            Host_Computer.StagingA_L2_ErrorCode := 0;
            Host_Computer.StagingA_L2_Retryable := FALSE;
            Host_Computer.StagingA_L2_CompletedSeq := Host_Computer.StagingA_L2_AcceptedSeq;
            Host_Computer.StagingA_L2_Step := 99;
            Host_Computer.StagingA_L2_State := 20;

        ELSE
            Host_Computer.StagingA_L2_ErrorCode := 103;
            Host_Computer.StagingA_L2_Retryable := FALSE;
            Host_Computer.StagingA_L2_CompletedSeq := Host_Computer.StagingA_L2_AcceptedSeq;
            Host_Computer.StagingA_L2_State := 40;
    END_CASE
END_IF

// 上位机看到终态后会清 Start=FALSE，并等待 State 回 IDLE。
// 保留 CompletedSeq，不清它，否则上位机会丢失已完成序号。
IF NOT Host_Computer.StagingA_L2_Start THEN
    IF (Host_Computer.StagingA_L2_State = 20)
    OR (Host_Computer.StagingA_L2_State = 30)
    OR (Host_Computer.StagingA_L2_State = 40)
    OR (Host_Computer.StagingA_L2_State = 50) THEN
        Host_Computer.StagingA_L2_State := 0;
        Host_Computer.StagingA_L2_ActiveCode := 0;
        Host_Computer.StagingA_L2_Step := 0;
        Host_Computer.StagingA_L2_ErrorCode := 0;
        Host_Computer.StagingA_L2_SafeState := 0;
        Host_Computer.StagingA_L2_Retryable := FALSE;
    END_IF
END_IF

END_PROGRAM

// Device/Application/50_action/Rail_L2
PROGRAM Rail_L2
VAR
	L2_StartTrig : R_TRIG;
	fTgt: LREAL;
END_VAR

(* 地轨 11Y L2 统一动作派发器 (第7通道).
   按位置码移地轨: Rail_L2_ActionCode=10 -> 移到 Rail_Pos_Target[Rail_Target_Position] (1..6, PC 真源).
   地轨坐标真源已收编为 PC 写的 Rail_Pos_Target[]; HMI position[] 降为手动示教工作副本, 自动不再读它.
   Start 上升沿接受 -> RUNNING 下发移动 -> bAbMoveDone=DONE. *)
L2_StartTrig(CLK := Rail_L2_Start);

(* Global deployment/startup gate: reject before any physical action is dispatched. *)
IF L2_StartTrig.Q AND (Rail_L2_State=0)
	AND ((NOT PLC_Ready) OR (PLC_Deploy_State<>0)) THEN
	Rail_L2_AcceptedSeq := Rail_L2_RequestSeq;
	Rail_L2_ActiveCode := Rail_L2_ActionCode;
	Rail_L2_ErrorCode := 190;
	Rail_L2_Retryable := TRUE;
	Rail_L2_CompletedSeq := Rail_L2_RequestSeq;
	Rail_L2_State := 30;
	RETURN;
END_IF

CASE Rail_L2_State OF
	0:  (* IDLE *)
		Rail_L2_Step := 0;
		IF L2_StartTrig.Q THEN
			Rail_L2_AcceptedSeq := Rail_L2_RequestSeq;
			Rail_L2_ActiveCode  := Rail_L2_ActionCode;
			Rail_L2_ErrorCode   := 0;
			Rail_L2_Retryable   := FALSE;
// 			IF Rail_L2_ActionCode = 10
// 			   AND Rail_Target_Position >= 1 AND Rail_Target_Position <= 6 THEN
// 				Rail_L2_SafeState := 0;
// // 				地轨轴11YDATE.fAbsTarget := HMI_地轨轴11Y.position[Rail_Target_Position];
// 				地轨轴11YDATE.fAbsTarget := Rail_Pos_Target[Rail_Target_Position];
// 				地轨轴11YDATE.xMoveAbs   := TRUE;
// 				Rail_L2_State := 10;   (* RUNNING *)
// 			ELSE
// 				Rail_L2_ErrorCode    := 101;  (* 未知动作码 / 非法位置码 *)
// 				Rail_L2_Retryable    := TRUE;
// 				Rail_L2_CompletedSeq := Rail_L2_AcceptedSeq;
// 				Rail_L2_State        := 30;   (* REJECTED *)
// 			END_IF
			IF Rail_L2_ActionCode = 10 AND Rail_Target_Position >= 1 AND Rail_Target_Position <= 6 THEN
				fTgt := Rail_Pos_Target[Rail_Target_Position];     (* PC 真源坐标 *)
				IF fTgt <= 0.0 OR fTgt > 3000.0 THEN
					(* 兜底: PC 未 push / 重启后 Rail_Pos_Target 归 0 / 越限 → 拒绝, 绝不移到 0 端 *)
					Rail_L2_ErrorCode    := 102;   (* 目标未初始化或越限 *)
					Rail_L2_Retryable    := TRUE;
					Rail_L2_CompletedSeq := Rail_L2_AcceptedSeq;
					Rail_L2_State        := 30;    (* REJECTED *)
				ELSE
					Rail_L2_SafeState        := 0;
					地轨轴11YDATE.fAbsTarget := fTgt;
					地轨轴11YDATE.xMoveAbs   := TRUE;
					Rail_L2_State            := 10; (* RUNNING *)
				END_IF
			ELSE
				Rail_L2_ErrorCode    := 101;   (* 未知动作码 / 非法位置码 *)
				Rail_L2_Retryable    := TRUE;
				Rail_L2_CompletedSeq := Rail_L2_AcceptedSeq;
				Rail_L2_State        := 30;    (* REJECTED *)
END_IF
		END_IF

	10: (* RUNNING *)
		IF Rail_L2_Reset THEN                 (* RUNNING 中 RESET: 中止回 IDLE *)
			地轨轴11YDATE.xMoveAbs := FALSE;
			Rail_L2_State := 0;
		ELSIF 地轨轴11YDATE.bAbMoveDone THEN
			地轨轴11YDATE.xMoveAbs   := FALSE;
			Rail_L2_CompletedSeq := Rail_L2_AcceptedSeq;
			Rail_L2_State        := 20;   (* DONE *)
		END_IF
		(* 如地轨伺服有报警位, 在此 ELSIF <报警> THEN 置 Rail_L2_ErrorCode + State:=40 *)

	20, 30, 40, 50:  (* 终态: 等 Start 落沿或 Reset 回 IDLE *)
		IF (NOT Rail_L2_Start) OR Rail_L2_Reset THEN
			Rail_L2_State := 0;
		END_IF
END_CASE

END_PROGRAM

// Device/Application/50_action/FeedLift_L2
PROGRAM FeedLift_L2
VAR
	初始化step: INT;
	上料step: INT;
	下料step: INT;
	bActionDone: BOOL;
	bActionError: BOOL;
	L2_StartTrig: R_TRIG;
	feedlift_TO: TON;
	FeedLift_1Z_RaiseRetryCount : INT;
	FeedLift_1Z_RaiseStartPos   : LREAL;
	FeedLift_1Z_ClearRetryCount : INT;
	FeedLift_1Z_ClearStartPos   : LREAL;
	FeedLift_2Z_ReadyRetryCount : INT;
	FeedLift_2Z_ReadyStartPos   : LREAL;
	FeedLift_2Z_BuryRetryCount  : INT;
	FeedLift_2Z_BuryStartPos    : LREAL;
END_VAR

(* FeedLift 工位 L2 统一动作派发器
   按 FeedLift_L2_ActionCode 派发到纯设备原子动作 (不含机器人/相机/CNC 握手).
   Start 上升沿接受请求 -> RUNNING 每周期调用对应原子 -> bActionDone=DONE / bActionError=ERROR. *)
L2_StartTrig(CLK := FeedLift_L2_Start);

(* Global deployment/startup gate: reject before any physical action is dispatched. *)
IF L2_StartTrig.Q AND (FeedLift_L2_State=0)
	AND ((NOT PLC_Ready) OR (PLC_Deploy_State<>0)) THEN
	FeedLift_L2_AcceptedSeq := FeedLift_L2_RequestSeq;
	FeedLift_L2_ActiveCode := FeedLift_L2_ActionCode;
	FeedLift_L2_ErrorCode := 190;
	FeedLift_L2_Retryable := TRUE;
	FeedLift_L2_CompletedSeq := FeedLift_L2_RequestSeq;
	FeedLift_L2_State := 30;
	RETURN;
END_IF

CASE FeedLift_L2_State OF
	0:  (* IDLE *)
		FeedLift_L2_Step := 0;
		IF L2_StartTrig.Q THEN
			FeedLift_L2_AcceptedSeq := FeedLift_L2_RequestSeq;
			FeedLift_L2_ActiveCode  := FeedLift_L2_ActionCode;
			FeedLift_L2_ErrorCode   := 0;
			FeedLift_L2_Retryable   := FALSE;
			bActionDone  := FALSE;
			bActionError := FALSE;
			初始化step := 0;
			上料step := 0;
			下料step := 0;
			CASE FeedLift_L2_ActionCode OF
				10, 11, 12, 13, 21, 22, 91:
					FeedLift_L2_SafeState := 0;
					FeedLift_L2_State     := 10;   (* RUNNING *)
			ELSE
				FeedLift_L2_ErrorCode    := 101;  (* 未知动作码 *)
				FeedLift_L2_Retryable    := TRUE;
				FeedLift_L2_CompletedSeq := FeedLift_L2_AcceptedSeq;
				FeedLift_L2_State        := 30;   (* REJECTED *)
			END_CASE
		END_IF

	10: (* RUNNING *)
		IF FeedLift_L2_Reset THEN FeedLift_L2_State := 0; RETURN; END_IF   (* RUNNING 中 RESET: 中止挂死动作 *)
		CASE FeedLift_L2_ActiveCode OF
			10: A10_init_初始化();
			11: A11_feed_raise();
			12: A12_feed_lower();
			13: A13_feed_clear();
			21: A21_unload_ready();
			22: A22_unload_bury();
			91: A91_endcheck();
		END_CASE
		IF bActionDone THEN
			bActionDone              := FALSE;
			FeedLift_L2_CompletedSeq := FeedLift_L2_AcceptedSeq;
			FeedLift_L2_State        := 20;   (* DONE *)
		ELSIF bActionError THEN              (* 设备预条件未满足 -> 报错交上位机 *)
			bActionError             := FALSE;
			FeedLift_L2_Retryable    := TRUE;
			FeedLift_L2_CompletedSeq := FeedLift_L2_AcceptedSeq;
			FeedLift_L2_State        := 40;   (* ERROR; ErrorCode 由原子置 *)
		END_IF

	20, 30, 40, 50:  (* 终态: 等 Start 落沿或 Reset 回 IDLE *)
		IF (NOT FeedLift_L2_Start) OR FeedLift_L2_Reset THEN
			FeedLift_L2_State := 0;
		END_IF
END_CASE

ACTION A11_feed_raise:
(* FeedLift feed_raise: bounded 1Z jog; final PE1 stable TRUE *)
// CASE 上料step OF
// 	0:
// 		Z1JOG_pos:=FALSE;
// 		feedlift_TO(IN:=FALSE, PT:=T#200MS);
// 		IF FeedLift_1Z_SearchLowTarget >= FeedLift_1Z_SearchHighTarget THEN
// 			FeedLift_L2_ErrorCode:=303;
// 			上料step:=0;
// 			bActionError:=TRUE;
// 		ELSIF 玻璃上料轴1ZDATE.bHomed AND 玻璃升降接近开关1 AND 上料进料传感器 AND NOT Alarm.0 THEN
// 			上料step:=10;
// 		ELSE
// 			feedlift_TO(IN:=TRUE, PT:=T#10S);
// 			IF feedlift_TO.Q THEN
// 				FeedLift_L2_ErrorCode:=301;
// 				上料step:=0;
// 				bActionError:=TRUE;
// 			END_IF
// 		END_IF
// 	10:
// 		feedlift_TO(IN:=FALSE, PT:=T#200MS);
// 		IF 玻璃升降光电开关1 THEN
// 			Z1JOG_pos:=FALSE;
// 			上料step:=20;
// 		ELSIF 玻璃上料轴1ZDATE.fActPos < FeedLift_1Z_SearchHighTarget THEN
// 			Z1JOG_pos:=TRUE;
// 		ELSE
// 			Z1JOG_pos:=FALSE;
// 			FeedLift_L2_ErrorCode:=304;
// 			上料step:=0;
// 			bActionError:=TRUE;
// 		END_IF
// 	20:
// 		Z1JOG_pos:=FALSE;
// 		feedlift_TO(IN:=玻璃升降光电开关1, PT:=T#200MS);
// 		IF feedlift_TO.Q THEN
// 			上料step:=0;
// 			bActionDone:=TRUE;
// 		ELSIF NOT 玻璃升降光电开关1 THEN
// 			IF 玻璃上料轴1ZDATE.fActPos < FeedLift_1Z_SearchHighTarget THEN
// 				上料step:=10;
// 			ELSE
// 				FeedLift_L2_ErrorCode:=304;
// 				上料step:=0;
// 				bActionError:=TRUE;
// 			END_IF
// 		END_IF
// END_CASE

(* FeedLift feed_raise:
   目标是找到并停在 1Z 上料取料位: 玻璃升降光电开关1 = TRUE。
   - 启动时已 TRUE: 原地停住, 稳定确认 DONE。
   - 启动时 FALSE: 只向上搜索 TRUE。
   - 看到 TRUE 后先停住, 再计时确认。
   - 确认中抖成 FALSE: 只向上小幅重捕获。
   - 失败用 304, 通过 FeedLift_L2_Step 区分阶段。 *)
CASE 上料step OF
	0:
		FeedLift_L2_Step := 11;  (* 初始化 / 前置检查 *)
		Z1JOG_pos := FALSE;
		feedlift_TO(IN := FALSE, PT := T#300MS);
		FeedLift_1Z_RaiseRetryCount := 0;
		FeedLift_1Z_RaiseStartPos := 玻璃上料轴1ZDATE.fActPos;

		IF FeedLift_1Z_SearchLowTarget >= FeedLift_1Z_SearchHighTarget THEN
			FeedLift_L2_ErrorCode := 303;
			上料step := 0;
			bActionError := TRUE;
		ELSE
			上料step := 5;
		END_IF

	5:
		FeedLift_L2_Step := 11;  (* 等待前置条件满足 *)
		Z1JOG_pos := FALSE;

		IF 玻璃上料轴1ZDATE.bHomed AND 玻璃升降接近开关1 AND 上料进料传感器 AND NOT Alarm.0 THEN
			feedlift_TO(IN := FALSE, PT := T#300MS);
			IF 玻璃升降光电开关1 THEN
				上料step := 20;
			ELSE
				上料step := 10;
			END_IF
		ELSE
			feedlift_TO(IN := TRUE, PT := T#10S);
			IF feedlift_TO.Q THEN
				FeedLift_L2_ErrorCode := 301;
				上料step := 0;
				bActionError := TRUE;
			END_IF
		END_IF

	10:
		FeedLift_L2_Step := 11;  (* 向上搜索 TRUE *)
		feedlift_TO(IN := FALSE, PT := T#300MS);

		IF 玻璃升降光电开关1 THEN
			Z1JOG_pos := FALSE;
			上料step := 20;
		ELSIF 玻璃上料轴1ZDATE.fActPos < FeedLift_1Z_SearchHighTarget THEN
			Z1JOG_pos := TRUE;
		ELSE
			Z1JOG_pos := FALSE;
			FeedLift_L2_Step := 14;  (* 失败收敛 *)
			FeedLift_L2_ErrorCode := 304;
			上料step := 0;
			bActionError := TRUE;
		END_IF

	20:
		FeedLift_L2_Step := 12;  (* 停住后确认 TRUE 稳定 *)
		Z1JOG_pos := FALSE;
		feedlift_TO(IN := 玻璃升降光电开关1, PT := T#300MS);

		IF feedlift_TO.Q THEN
			上料step := 0;
			bActionDone := TRUE;
		ELSIF NOT 玻璃升降光电开关1 THEN
			feedlift_TO(IN := FALSE, PT := T#300MS);
			IF FeedLift_1Z_RaiseRetryCount < 2 THEN
				FeedLift_1Z_RaiseRetryCount := FeedLift_1Z_RaiseRetryCount + 1;
				FeedLift_1Z_RaiseStartPos := 玻璃上料轴1ZDATE.fActPos;
				上料step := 30;
			ELSE
				FeedLift_L2_Step := 14;  (* 失败收敛 *)
				FeedLift_L2_ErrorCode := 304;
				上料step := 0;
				bActionError := TRUE;
			END_IF
		END_IF

	30:
		FeedLift_L2_Step := 13;  (* 小幅向上重捕获 TRUE *)
		feedlift_TO(IN := FALSE, PT := T#300MS);

		IF 玻璃升降光电开关1 THEN
			Z1JOG_pos := FALSE;
			上料step := 20;
		ELSIF 玻璃上料轴1ZDATE.fActPos >= FeedLift_1Z_SearchHighTarget THEN
			Z1JOG_pos := FALSE;
			FeedLift_L2_Step := 14;  (* 失败收敛 *)
			FeedLift_L2_ErrorCode := 304;
			上料step := 0;
			bActionError := TRUE;
		ELSIF (玻璃上料轴1ZDATE.fActPos - FeedLift_1Z_RaiseStartPos) >= 2.0 THEN
			Z1JOG_pos := FALSE;
			FeedLift_L2_Step := 14;  (* 失败收敛 *)
			FeedLift_L2_ErrorCode := 304;
			上料step := 0;
			bActionError := TRUE;
		ELSE
			Z1JOG_pos := TRUE;
		END_IF
END_CASE
END_ACTION

ACTION A10_init_初始化:
(* FeedLift init:
   清 L2 域内的残留命令位, 再校验 1Z/2Z 已回零。
   - jog 位: 任一搜索动作被 L2_Reset 中止时会停在 TRUE, 不清则下次上电即自行走轴。
   - xMoveRel: A12_feed_lower 在 step0 置位、step10 才清, 中途 Reset 同样留 TRUE。
   - 步序变量由派发器 IDLE 受理时统一清零, 此处不重复。
   本动作不产生任何轴运动: 双轴回零只能在 HMI 按【一键回原点】, 上位机无此通道,
   故未回零时只报 308 交上位机, 不自行 Home。
   失败用 308, 通过 FeedLift_L2_Step 区分阶段。 *)
CASE 初始化step OF
	0:
		FeedLift_L2_Step := 51;  (* 清残留命令位 *)
		Z1JOG_pos := FALSE;
		Z1JOG_neg := FALSE;
		Z2JOG_POS := FALSE;
		Z2JOG_NEG := FALSE;
		玻璃上料轴1ZDATE.xMoveRel := FALSE;
		玻璃上料轴2ZDATE.xMoveRel := FALSE;
		feedlift_TO(IN := FALSE, PT := T#300MS);
		初始化step := 10;

	10:
		FeedLift_L2_Step := 52;  (* 校验双轴已回零 *)
		IF 玻璃上料轴1ZDATE.bHomed AND 玻璃上料轴2ZDATE.bHomed THEN
			初始化step := 0;
			bActionDone := TRUE;
		ELSE
			feedlift_TO(IN := TRUE, PT := T#5S);
			IF feedlift_TO.Q THEN
				FeedLift_L2_Step := 54;  (* 失败收敛 *)
				FeedLift_L2_ErrorCode := 308;
				初始化step := 0;
				bActionError := TRUE;
			END_IF
		END_IF
END_CASE
END_ACTION

ACTION A22_unload_bury:
(* FeedLift unload_bury: bounded 2Z jog to make PE2 stable FALSE; reverse once if low misses *)
// CASE 下料step OF
// 	0:
// 		Z2JOG_POS:=FALSE;
// 		Z2JOG_NEG:=FALSE;
// 		feedlift_TO(IN:=FALSE, PT:=T#200MS);
// 		IF FeedLift_2Z_SearchLowTarget >= FeedLift_2Z_SearchHighTarget THEN
// 			FeedLift_L2_ErrorCode:=303;
// 			下料step:=0;
// 			bActionError:=TRUE;
// 		ELSIF 玻璃升降光电开关2 AND 玻璃升降接近开关2 THEN
// 			下料step:=10;
// 		ELSE
// 			feedlift_TO(IN:=TRUE, PT:=T#10S);
// 			IF feedlift_TO.Q THEN
// 				FeedLift_L2_ErrorCode:=302;
// 				下料step:=0;
// 				bActionError:=TRUE;
// 			END_IF
// 		END_IF
// 	10:
// 		Z2JOG_POS:=FALSE;
// 		IF NOT 玻璃升降光电开关2 THEN
// 			Z2JOG_NEG:=FALSE;
// 			下料step:=30;
// 		ELSIF 玻璃上料轴2ZDATE.fActPos > FeedLift_2Z_SearchLowTarget THEN
// 			Z2JOG_NEG:=TRUE;
// 		ELSE
// 			Z2JOG_NEG:=FALSE;
// 			下料step:=20;
// 		END_IF
// 	20:
// 		Z2JOG_NEG:=FALSE;
// 		IF NOT 玻璃升降光电开关2 THEN
// 			Z2JOG_POS:=FALSE;
// 			下料step:=30;
// 		ELSIF 玻璃上料轴2ZDATE.fActPos < FeedLift_2Z_SearchHighTarget THEN
// 			Z2JOG_POS:=TRUE;
// 		ELSE
// 			Z2JOG_POS:=FALSE;
// 			FeedLift_L2_ErrorCode:=305;
// 			下料step:=0;
// 			bActionError:=TRUE;
// 		END_IF
// 	30:
// 		Z2JOG_POS:=FALSE;
// 		Z2JOG_NEG:=FALSE;
// 		feedlift_TO(IN:=NOT 玻璃升降光电开关2, PT:=T#200MS);
// 		IF feedlift_TO.Q THEN
// 			下料step:=0;
// 			bActionDone:=TRUE;
// 		ELSIF 玻璃升降光电开关2 THEN
// 			IF 玻璃上料轴2ZDATE.fActPos > FeedLift_2Z_SearchLowTarget THEN
// 				下料step:=10;
// 			ELSIF 玻璃上料轴2ZDATE.fActPos < FeedLift_2Z_SearchHighTarget THEN
// 				下料step:=20;
// 			ELSE
// 				FeedLift_L2_ErrorCode:=305;
// 				下料step:=0;
// 				bActionError:=TRUE;
// 			END_IF
// 		END_IF
// END_CASE

(* FeedLift unload_bury:
   目标是机器人放废板后, 2Z 向下埋料直到 玻璃升降光电开关2 = FALSE。
   - 启动时已 FALSE: 原地停住, 稳定确认 DONE。
   - 启动时 TRUE: 只向下搜索 FALSE。
   - 看到 FALSE 后先停住, 再计时确认。
   - 确认中抖成 TRUE: 只向下小幅重捕获, 不反向上扫。
   - 失败用 305, 通过 FeedLift_L2_Step 区分阶段。 *)
CASE 下料step OF
	0:
		FeedLift_L2_Step := 31;  (* 初始化 / 前置检查 *)
		Z2JOG_POS := FALSE;
		Z2JOG_NEG := FALSE;
		feedlift_TO(IN := FALSE, PT := T#300MS);
		FeedLift_2Z_BuryRetryCount := 0;
		FeedLift_2Z_BuryStartPos := 玻璃上料轴2ZDATE.fActPos;

		IF FeedLift_2Z_SearchLowTarget >= FeedLift_2Z_SearchHighTarget THEN
			FeedLift_L2_ErrorCode := 303;
			下料step := 0;
			bActionError := TRUE;
		ELSE
			下料step := 5;
		END_IF

	5:
		FeedLift_L2_Step := 31;  (* 等待前置条件满足 *)
		Z2JOG_POS := FALSE;
		Z2JOG_NEG := FALSE;

		IF 玻璃上料轴2ZDATE.bHomed AND 玻璃升降接近开关2 AND NOT Alarm.1 THEN
			feedlift_TO(IN := FALSE, PT := T#300MS);
			IF NOT 玻璃升降光电开关2 THEN
				下料step := 20;
			ELSE
				下料step := 10;
			END_IF
		ELSE
			feedlift_TO(IN := TRUE, PT := T#10S);
			IF feedlift_TO.Q THEN
				FeedLift_L2_ErrorCode := 302;
				下料step := 0;
				bActionError := TRUE;
			END_IF
		END_IF

	10:
		FeedLift_L2_Step := 31;  (* 向下搜索 FALSE *)
		Z2JOG_POS := FALSE;
		feedlift_TO(IN := FALSE, PT := T#300MS);

		IF NOT 玻璃升降光电开关2 THEN
			Z2JOG_NEG := FALSE;
			下料step := 20;
		ELSIF 玻璃上料轴2ZDATE.fActPos > FeedLift_2Z_SearchLowTarget THEN
			Z2JOG_NEG := TRUE;
		ELSE
			Z2JOG_NEG := FALSE;
			FeedLift_L2_Step := 34;  (* 失败收敛 *)
			FeedLift_L2_ErrorCode := 305;
			下料step := 0;
			bActionError := TRUE;
		END_IF

	20:
		FeedLift_L2_Step := 32;  (* 停住后确认 FALSE 稳定 *)
		Z2JOG_POS := FALSE;
		Z2JOG_NEG := FALSE;
		feedlift_TO(IN := NOT 玻璃升降光电开关2, PT := T#300MS);

		IF feedlift_TO.Q THEN
			下料step := 0;
			bActionDone := TRUE;
		ELSIF 玻璃升降光电开关2 THEN
			feedlift_TO(IN := FALSE, PT := T#300MS);
			IF FeedLift_2Z_BuryRetryCount < 2 THEN
				FeedLift_2Z_BuryRetryCount := FeedLift_2Z_BuryRetryCount + 1;
				FeedLift_2Z_BuryStartPos := 玻璃上料轴2ZDATE.fActPos;
				下料step := 30;
			ELSE
				FeedLift_L2_Step := 34;  (* 失败收敛 *)
				FeedLift_L2_ErrorCode := 305;
				下料step := 0;
				bActionError := TRUE;
			END_IF
		END_IF

	30:
		FeedLift_L2_Step := 33;  (* 小幅向下重捕获 FALSE *)
		Z2JOG_POS := FALSE;
		feedlift_TO(IN := FALSE, PT := T#300MS);

		IF NOT 玻璃升降光电开关2 THEN
			Z2JOG_NEG := FALSE;
			下料step := 20;
		ELSIF 玻璃上料轴2ZDATE.fActPos <= FeedLift_2Z_SearchLowTarget THEN
			Z2JOG_NEG := FALSE;
			FeedLift_L2_Step := 34;  (* 失败收敛 *)
			FeedLift_L2_ErrorCode := 305;
			下料step := 0;
			bActionError := TRUE;
		ELSIF (FeedLift_2Z_BuryStartPos - 玻璃上料轴2ZDATE.fActPos) >= 2.0 THEN
			Z2JOG_NEG := FALSE;
			FeedLift_L2_Step := 34;  (* 失败收敛 *)
			FeedLift_L2_ErrorCode := 305;
			下料step := 0;
			bActionError := TRUE;
		ELSE
			Z2JOG_NEG := TRUE;
		END_IF
END_CASE
END_ACTION

ACTION A91_endcheck:
(* DEBUG: no-jog photoelectric stable-state confirmation *)
FeedLift_L2_Step := 91;
CASE FeedLift_DebugAxis OF
	1:
		feedlift_TO(IN:=(玻璃升降光电开关1 = FeedLift_DebugExpectedFinal), PT:=T#200MS);
		IF feedlift_TO.Q THEN bActionDone:=TRUE; END_IF
	2:
		feedlift_TO(IN:=(玻璃升降光电开关2 = FeedLift_DebugExpectedFinal), PT:=T#200MS);
		IF feedlift_TO.Q THEN bActionDone:=TRUE; END_IF
ELSE
	FeedLift_L2_ErrorCode:=306;
	bActionError:=TRUE;
END_CASE
END_ACTION

ACTION A13_feed_clear:
(* FeedLift feed_clear:
   目标是把 1Z 降到 玻璃升降光电开关1 = FALSE, 给随后的 feed_raise 让出"从 FALSE 侧逼近"的行程。
   - 启动时已 FALSE: 原地停住, 稳定确认 DONE。
   - 启动时 TRUE: 只向下搜索 FALSE。
   - 看到 FALSE 后先停住, 再计时确认。
   - 确认中抖回 TRUE: 只向下小幅重捕获, 不反向上扫。
   - 失败用 307, 通过 FeedLift_L2_Step 区分阶段。
   前置刻意不查 上料进料传感器: 本动作是向下退让给测量让位, 不该被仓内有无料卡住
   (空仓标定第一组正需要它能跑)。 *)
CASE 上料step OF
	0:
		FeedLift_L2_Step := 41;  (* 初始化 / 前置检查 *)
		Z1JOG_pos := FALSE;
		Z1JOG_neg := FALSE;
		feedlift_TO(IN := FALSE, PT := T#300MS);
		FeedLift_1Z_ClearRetryCount := 0;
		FeedLift_1Z_ClearStartPos := 玻璃上料轴1ZDATE.fActPos;

		IF FeedLift_1Z_SearchLowTarget >= FeedLift_1Z_SearchHighTarget THEN
			FeedLift_L2_ErrorCode := 303;
			上料step := 0;
			bActionError := TRUE;
		ELSE
			上料step := 5;
		END_IF

	5:
		FeedLift_L2_Step := 41;  (* 等待前置条件满足 *)
		Z1JOG_pos := FALSE;
		Z1JOG_neg := FALSE;

		IF 玻璃上料轴1ZDATE.bHomed AND 玻璃升降接近开关1 AND NOT Alarm.0 THEN
			feedlift_TO(IN := FALSE, PT := T#300MS);
			IF NOT 玻璃升降光电开关1 THEN
				上料step := 20;
			ELSE
				上料step := 10;
			END_IF
		ELSE
			feedlift_TO(IN := TRUE, PT := T#10S);
			IF feedlift_TO.Q THEN
				FeedLift_L2_ErrorCode := 301;
				上料step := 0;
				bActionError := TRUE;
			END_IF
		END_IF

	10:
		FeedLift_L2_Step := 41;  (* 向下搜索 FALSE *)
		Z1JOG_pos := FALSE;
		feedlift_TO(IN := FALSE, PT := T#300MS);

		IF NOT 玻璃升降光电开关1 THEN
			Z1JOG_neg := FALSE;
			上料step := 20;
		ELSIF 玻璃上料轴1ZDATE.fActPos > FeedLift_1Z_SearchLowTarget THEN
			Z1JOG_neg := TRUE;
		ELSE
			Z1JOG_neg := FALSE;
			FeedLift_L2_Step := 44;  (* 失败收敛 *)
			FeedLift_L2_ErrorCode := 307;
			上料step := 0;
			bActionError := TRUE;
		END_IF

	20:
		FeedLift_L2_Step := 42;  (* 停住后确认 FALSE 稳定 *)
		Z1JOG_pos := FALSE;
		Z1JOG_neg := FALSE;
		feedlift_TO(IN := NOT 玻璃升降光电开关1, PT := T#300MS);

		IF feedlift_TO.Q THEN
			上料step := 0;
			bActionDone := TRUE;
		ELSIF 玻璃升降光电开关1 THEN
			feedlift_TO(IN := FALSE, PT := T#300MS);
			IF FeedLift_1Z_ClearRetryCount < 2 THEN
				FeedLift_1Z_ClearRetryCount := FeedLift_1Z_ClearRetryCount + 1;
				FeedLift_1Z_ClearStartPos := 玻璃上料轴1ZDATE.fActPos;
				上料step := 30;
			ELSE
				FeedLift_L2_Step := 44;  (* 失败收敛 *)
				FeedLift_L2_ErrorCode := 307;
				上料step := 0;
				bActionError := TRUE;
			END_IF
		END_IF

	30:
		FeedLift_L2_Step := 43;  (* 小幅向下重捕获 FALSE *)
		Z1JOG_pos := FALSE;
		feedlift_TO(IN := FALSE, PT := T#300MS);

		IF NOT 玻璃升降光电开关1 THEN
			Z1JOG_neg := FALSE;
			上料step := 20;
		ELSIF 玻璃上料轴1ZDATE.fActPos <= FeedLift_1Z_SearchLowTarget THEN
			Z1JOG_neg := FALSE;
			FeedLift_L2_Step := 44;  (* 失败收敛 *)
			FeedLift_L2_ErrorCode := 307;
			上料step := 0;
			bActionError := TRUE;
		ELSIF (FeedLift_1Z_ClearStartPos - 玻璃上料轴1ZDATE.fActPos) >= 2.0 THEN
			Z1JOG_neg := FALSE;
			FeedLift_L2_Step := 44;  (* 失败收敛 *)
			FeedLift_L2_ErrorCode := 307;
			上料step := 0;
			bActionError := TRUE;
		ELSE
			Z1JOG_neg := TRUE;
		END_IF
END_CASE
END_ACTION

ACTION A12_feed_lower:
(* 上料: 机器人吸住玻璃后, Z1 相对下降 5mm 让位 *)
CASE 上料step OF
	0:
		玻璃上料轴1ZDATE.fRelTarget:=-5.0;
		玻璃上料轴1ZDATE.xMoveRel:=TRUE;
		上料step:=10;
	10:
		IF 玻璃上料轴1ZDATE.bReMoveDone THEN
			玻璃上料轴1ZDATE.xMoveRel:=FALSE;
			上料step:=0;
			bActionDone:=TRUE;
		END_IF
END_CASE
END_ACTION

ACTION A21_unload_ready:
(* FeedLift unload_ready: bounded 2Z search PE2 then leave until PE2 stable FALSE *)
// CASE 下料step OF
// 	0:
// 		Z2JOG_POS:=FALSE;
// 		Z2JOG_NEG:=FALSE;
// 		feedlift_TO(IN:=FALSE, PT:=T#200MS);
// 		IF FeedLift_2Z_SearchLowTarget >= FeedLift_2Z_SearchHighTarget THEN
// 			FeedLift_L2_ErrorCode:=303;
// 			下料step:=0;
// 			bActionError:=TRUE;
// 		ELSIF 玻璃上料轴2ZDATE.bHomed AND 下料出料传感器 AND NOT Alarm.1 THEN
// 			IF 玻璃升降光电开关2 THEN
// 				下料step:=20;
// 			ELSE
// 				下料step:=10;
// 			END_IF
// 		ELSE
// 			feedlift_TO(IN:=TRUE, PT:=T#10S);
// 			IF feedlift_TO.Q THEN
// 				FeedLift_L2_ErrorCode:=302;
// 				下料step:=0;
// 				bActionError:=TRUE;
// 			END_IF
// 		END_IF
// 	10:
// 		feedlift_TO(IN:=FALSE, PT:=T#200MS);
// 		Z2JOG_NEG:=FALSE;
// 		IF 玻璃升降光电开关2 THEN
// 			Z2JOG_POS:=FALSE;
// 			下料step:=20;
// 		ELSIF 玻璃上料轴2ZDATE.fActPos < FeedLift_2Z_SearchHighTarget THEN
// 			Z2JOG_POS:=TRUE;
// 		ELSE
// 			Z2JOG_POS:=FALSE;
// 			FeedLift_L2_ErrorCode:=305;
// 			下料step:=0;
// 			bActionError:=TRUE;
// 		END_IF
// 	20:
// 		Z2JOG_POS:=FALSE;
// 		IF NOT 玻璃升降光电开关2 THEN
// 			Z2JOG_NEG:=FALSE;
// 			下料step:=30;
// 		ELSIF 玻璃上料轴2ZDATE.fActPos > FeedLift_2Z_SearchLowTarget THEN
// 			Z2JOG_NEG:=TRUE;
// 		ELSE
// 			Z2JOG_NEG:=FALSE;
// 			FeedLift_L2_ErrorCode:=305;
// 			下料step:=0;
// 			bActionError:=TRUE;
// 		END_IF
// 	30:
// 		Z2JOG_POS:=FALSE;
// 		Z2JOG_NEG:=FALSE;
// 		feedlift_TO(IN:=NOT 玻璃升降光电开关2, PT:=T#200MS);
// 		IF feedlift_TO.Q THEN
// 			下料step:=0;
// 			bActionDone:=TRUE;
// 		ELSIF 玻璃升降光电开关2 THEN
// 			IF 玻璃上料轴2ZDATE.fActPos > FeedLift_2Z_SearchLowTarget THEN
// 				下料step:=20;
// 			ELSE
// 				FeedLift_L2_ErrorCode:=305;
// 				下料step:=0;
// 				bActionError:=TRUE;
// 			END_IF
// 		END_IF
// END_CASE

(* FeedLift unload_ready:
   目标是找到并停在 2Z 废料接料位: 玻璃升降光电开关2 = TRUE。
   - 启动时已 TRUE: 原地停住, 稳定确认 DONE。
   - 启动时 FALSE: 只向上搜索 TRUE。
   - 看到 TRUE 后先停住, 再计时确认。
   - 确认中抖成 FALSE: 只向上小幅重捕获, 不向下搜索。
   - 失败统一报 305, 通过 FeedLift_L2_Step 区分阶段。 *)
(* FeedLift unload_ready:
   目标是找到并停在 2Z 废料接料位: 玻璃升降光电开关2 = TRUE。
   - 启动时已 TRUE: 原地停住, 稳定确认 DONE。
   - 启动时 FALSE: 只向上搜索 TRUE。
   - 看到 TRUE 后先停住, 再计时确认。
   - 确认中抖成 FALSE: 只向上小幅重捕获, 不向下搜索。
   - 失败统一报 305, 通过 FeedLift_L2_Step 区分阶段。 *)
CASE 下料step OF
	0:
		FeedLift_L2_Step := 21;  (* 初始化 / 前置检查 *)
		Z2JOG_POS := FALSE;
		Z2JOG_NEG := FALSE;
		feedlift_TO(IN := FALSE, PT := T#300MS);
		FeedLift_2Z_ReadyRetryCount := 0;
		FeedLift_2Z_ReadyStartPos := 玻璃上料轴2ZDATE.fActPos;

		IF FeedLift_2Z_SearchLowTarget >= FeedLift_2Z_SearchHighTarget THEN
			FeedLift_L2_ErrorCode := 303;
			下料step := 0;
			bActionError := TRUE;
		ELSE
			下料step := 5;
		END_IF

	5:
		FeedLift_L2_Step := 21;  (* 等待前置条件满足 *)
		Z2JOG_POS := FALSE;
		Z2JOG_NEG := FALSE;

		IF 玻璃上料轴2ZDATE.bHomed AND 下料出料传感器 AND NOT Alarm.1 THEN
			feedlift_TO(IN := FALSE, PT := T#300MS);
			IF 玻璃升降光电开关2 THEN
				下料step := 20;
			ELSE
				下料step := 10;
			END_IF
		ELSE
			feedlift_TO(IN := TRUE, PT := T#10S);
			IF feedlift_TO.Q THEN
				FeedLift_L2_ErrorCode := 302;
				下料step := 0;
				bActionError := TRUE;
			END_IF
		END_IF

	10:
		FeedLift_L2_Step := 21;  (* 向上搜索 TRUE *)
		Z2JOG_NEG := FALSE;
		feedlift_TO(IN := FALSE, PT := T#300MS);

		IF 玻璃升降光电开关2 THEN
			Z2JOG_POS := FALSE;
			下料step := 20;
		ELSIF 玻璃上料轴2ZDATE.fActPos < FeedLift_2Z_SearchHighTarget THEN
			Z2JOG_POS := TRUE;
		ELSE
			Z2JOG_POS := FALSE;
			FeedLift_L2_Step := 24;  (* 失败收敛 *)
			FeedLift_L2_ErrorCode := 305;
			下料step := 0;
			bActionError := TRUE;
		END_IF

	20:
		FeedLift_L2_Step := 22;  (* 停住后确认 TRUE 稳定 *)
		Z2JOG_POS := FALSE;
		Z2JOG_NEG := FALSE;
		feedlift_TO(IN := 玻璃升降光电开关2, PT := T#300MS);

		IF feedlift_TO.Q THEN
			下料step := 0;
			bActionDone := TRUE;
		ELSIF NOT 玻璃升降光电开关2 THEN
			feedlift_TO(IN := FALSE, PT := T#300MS);
			IF FeedLift_2Z_ReadyRetryCount < 2 THEN
				FeedLift_2Z_ReadyRetryCount := FeedLift_2Z_ReadyRetryCount + 1;
				FeedLift_2Z_ReadyStartPos := 玻璃上料轴2ZDATE.fActPos;
				下料step := 30;
			ELSE
				FeedLift_L2_Step := 24;  (* 失败收敛 *)
				FeedLift_L2_ErrorCode := 305;
				下料step := 0;
				bActionError := TRUE;
			END_IF
		END_IF

	30:
		FeedLift_L2_Step := 23;  (* 小幅向上重捕获 TRUE *)
		Z2JOG_NEG := FALSE;
		feedlift_TO(IN := FALSE, PT := T#300MS);

		IF 玻璃升降光电开关2 THEN
			Z2JOG_POS := FALSE;
			下料step := 20;
		ELSIF 玻璃上料轴2ZDATE.fActPos >= FeedLift_2Z_SearchHighTarget THEN
			Z2JOG_POS := FALSE;
			FeedLift_L2_Step := 24;  (* 失败收敛 *)
			FeedLift_L2_ErrorCode := 305;
			下料step := 0;
			bActionError := TRUE;
		ELSIF (玻璃上料轴2ZDATE.fActPos - FeedLift_2Z_ReadyStartPos) >= 2.0 THEN
			Z2JOG_POS := FALSE;
			FeedLift_L2_Step := 24;  (* 失败收敛 *)
			FeedLift_L2_ErrorCode := 305;
			下料step := 0;
			bActionError := TRUE;
		ELSE
			Z2JOG_POS := TRUE;
		END_IF
END_CASE
END_ACTION

END_PROGRAM

// Device/Application/50_action/Sampling_L2
PROGRAM Sampling_L2
VAR
	初始化step: INT;
	清洗step: INT;
	清洗计数: INT;
	放硅胶板STEP: INT;
	上样准备step: INT;
	吸收液体step: INT;
	rinse_mix_step: INT;
	rinse_mix_cycle: INT;
	点样step: INT;
	喷涂移轴step: INT;
	N: INT;
	A: INT;
	打样伺服移动step: INT;
	spot_band_step: INT;
	spot_band_dry_count: INT;
	spot_band_old_6x_velocity: LREAL;
	spot_band_velocity_saved: BOOL;
	spot_band_q_sent: BOOL;
	spot_band_pB: POINTER TO BYTE;
	spot_band_pos: INT;
	spot_band_pos_valid: BOOL;
	spot_band_k: INT;
	spot_band_pass_count: INT;
	spot_band_query_retry: INT;
	spot_band_dir: BOOL;
	spot_band_query_active: BOOL;
	spot_band_query_done: BOOL;
	sample_q_sent: BOOL;
	sample_pB: POINTER TO BYTE;
	sample_pos: INT;
	sample_pos_valid: BOOL;
	sample_k: WORD;
	sample_query_retry: INT;
	sample_relative_steps: INT;
	sample_relative_valid: BOOL;
	// A50 移孔位前的气隔断吸气段 (Sampling_sample_instructions[2]); 专用实例, 不占 TON/R_TRIG 数组
	sample_gap_wait: TON;
	sample_gap_idle: R_TRIG;
	bActionDone: BOOL;
	bActionError: BOOL;
	TON_0: TON;
	TON_1: TON;
	rinse_mix_wait: TON;
	rinse_mix_idle: R_TRIG;
	L2_StartTrig: R_TRIG;
	R_TRIG: ARRAY[1..12] OF R_TRIG;
	TON: ARRAY[1..11] OF TON;
END_VAR

(* Sampling 工位 L2 统一动作派发器
   按 Sampling_L2_ActionCode 派发到纯设备原子动作 (不含机器人/相机/CNC 握手).
   Start 上升沿接受请求 -> RUNNING 每周期调用对应原子 -> bActionDone=DONE / bActionError=ERROR. *)
L2_StartTrig(CLK := Sampling_L2_Start);

(* Global deployment/startup gate: reject before any physical action is dispatched. *)
IF L2_StartTrig.Q AND (Sampling_L2_State=0)
	AND ((NOT PLC_Ready) OR (PLC_Deploy_State<>0)) THEN
	Sampling_L2_AcceptedSeq := Sampling_L2_RequestSeq;
	Sampling_L2_ActiveCode := Sampling_L2_ActionCode;
	Sampling_L2_ErrorCode := 190;
	Sampling_L2_Retryable := TRUE;
	Sampling_L2_CompletedSeq := Sampling_L2_RequestSeq;
	Sampling_L2_State := 30;
	RETURN;
END_IF

CASE Sampling_L2_State OF
	0:  (* IDLE *)
		Sampling_L2_Step := 0;
		IF L2_StartTrig.Q THEN
			Sampling_L2_AcceptedSeq := Sampling_L2_RequestSeq;
			Sampling_L2_ActiveCode  := Sampling_L2_ActionCode;
			Sampling_L2_ErrorCode   := 0;
			Sampling_L2_Retryable   := FALSE;
			bActionDone  := FALSE;
			bActionError := FALSE;
			初始化step := 0;
			清洗step := 0;
			放硅胶板STEP := 0;
			上样准备step := 0;
			吸收液体step := 0;
			rinse_mix_step := 0;
			rinse_mix_cycle := 0;
			点样step := 0;
			喷涂移轴step := 0;
			spot_band_step := 0;
			spot_band_dry_count := 0;
			spot_band_velocity_saved := FALSE;
			spot_band_query_active := FALSE;
			spot_band_query_done := FALSE;
			CASE Sampling_L2_ActionCode OF
				10, 20, 31, 32, 33, 40, 50, 55, 60, 61, 62:
					Sampling_L2_SafeState := 0;
					Sampling_L2_State     := 10;   (* RUNNING *)
			ELSE
				Sampling_L2_ErrorCode    := 101;  (* 未知动作码 *)
				Sampling_L2_Retryable    := TRUE;
				Sampling_L2_CompletedSeq := Sampling_L2_AcceptedSeq;
				Sampling_L2_State        := 30;   (* REJECTED *)
			END_CASE
		END_IF

	10: (* RUNNING *)
		IF Sampling_L2_Reset THEN
			IF Sampling_L2_ActiveCode = 55 THEN
				(* A55 非幂等动作：先撤销轴运动，等待串口空闲后发泵停止，再进入 INTERRUPTED。 *)
				上样轴5Z轴DATE.xMoveAbs := FALSE;
				上样轴4X轴DATE.xMoveAbs := FALSE;
				打样瓶上料轴3YDATE.xMoveAbs := FALSE;
				上样点样三通电池阀自动 := FALSE;
				rinse_mix_step := 0;
				rinse_mix_cycle := 0;
				IF %MW1300 = 0 THEN
					转发转存 := '/4T$R';
					%MW1300 := LEN(STR := 转发转存);
					泵站位符 := FALSE;
					Sampling_L2_Retryable := FALSE;
					Sampling_L2_CompletedSeq := Sampling_L2_AcceptedSeq;
					Sampling_L2_State := 50;  (* INTERRUPTED *)
				END_IF
				RETURN;
			END_IF
			IF (Sampling_L2_ActiveCode = 20) OR (Sampling_L2_ActiveCode = 40) OR
			   (Sampling_L2_ActiveCode = 50) OR (Sampling_L2_ActiveCode = 60) OR
			   (Sampling_L2_ActiveCode = 62) THEN
				泵站位符 := FALSE;
			END_IF
			IF Sampling_L2_ActiveCode = 62 THEN
				上样点样三通电池阀自动 := FALSE;
				上样吹气自动 := FALSE;
				点样轴6XDATE.xMoveAbs := FALSE;
				点样轴7YDATE.xMoveAbs := FALSE;
				IF spot_band_velocity_saved THEN
					点样轴6XDATE.fVelocity := spot_band_old_6x_velocity;
					spot_band_velocity_saved := FALSE;
				END_IF
				spot_band_step := 0;
				spot_band_query_active := FALSE;
				spot_band_query_done := FALSE;
			END_IF
			Sampling_L2_State := 0;
			RETURN;
		END_IF
		CASE Sampling_L2_ActiveCode OF
			10: A10_init_初始化();
			20: A20_clean_清洗();
			31: A31_放板移轴();
			32: A32_放板定位();
			33: A33_定位松开();
			40: A40_prep_上样准备();
			50: A50_absorb_吸收液体();
			55: A55_润洗吹打混匀();
			60: A60_spray_点样();
			61: A61_喷涂移轴();
			62: A62_单条带点样();
		END_CASE
		IF bActionDone THEN
			bActionDone              := FALSE;
			Sampling_L2_CompletedSeq := Sampling_L2_AcceptedSeq;
			Sampling_L2_State        := 20;   (* DONE *)
		ELSIF bActionError THEN              (* 设备预条件未满足 -> 报错交上位机 *)
			bActionError             := FALSE;
			Sampling_L2_Retryable    := (Sampling_L2_ErrorCode <> 466);
			Sampling_L2_CompletedSeq := Sampling_L2_AcceptedSeq;
			Sampling_L2_State        := 40;   (* ERROR; ErrorCode 由原子置 *)
		END_IF

	20, 30, 40:  (* DONE/REJECTED/ERROR：等 Start 落沿或 Reset 回 IDLE *)
		IF (NOT Sampling_L2_Start) OR Sampling_L2_Reset THEN
			Sampling_L2_State := 0;
		END_IF

	50:  (* INTERRUPTED：Reset 与 Start 均撤销后才回 IDLE，避免中断态被同一扫描吞掉。 *)
		IF (NOT Sampling_L2_Start) AND (NOT Sampling_L2_Reset) THEN
			Sampling_L2_State := 0;
		END_IF
END_CASE

ACTION A33_定位松开:
(* 定位松开: 松开上样定位气缸释放硅胶板 (上位机随后驱动机器人取板); 镜像 A32 放板定位 *)
上样定位自动 := FALSE;
bActionDone := TRUE;
END_ACTION

ACTION A50_absorb_吸收液体:
(* 吸收液体: Z回零->[空气中吸气隔断]->XY->Z下探->查询真活塞位->行程校验->P<n>相对回抽->Z回零
   气隔断 (指令[2], 绝对 A{gap}) 必须在移向孔位【之前】于原位空气中吸入:
   吸气前针尖内为满液, 带液移动途中的挂壁滴液会滴进样品孔稀释样品; 吸气后针尖端为空气段才安全移动。
   [2] 为空串时整段跳过 (兼容编排先调 A40_prep 建立气隔断的旧路径)。
   绝对语义使润洗轮天然幂等: A55 终态活塞已在 A{gap}, 再绝对吸至 A{gap} 为零位移。 *)
TON_0(IN:=吸收液体step=30, PT:=T#0.5S);
TON_1(IN:=NOT 点样气泡传感器, PT:=T#5S);
TON[11](IN:=sample_q_sent, PT:=T#200MS);
R_TRIG[10](CLK:=%MX2005.5);
sample_gap_wait(IN:=吸收液体step=3, PT:=T#0.5S);
sample_gap_idle(CLK:=%MX2005.5);
IF TRUE THEN
	CASE 吸收液体step OF
		0:
			上样轴5Z轴DATE.fAbsTarget:=0;
			上样轴5Z轴DATE.xMoveAbs:=TRUE;
			IF 上样轴5Z轴DATE.bAbMoveDone THEN
				上样轴5Z轴DATE.xMoveAbs:=FALSE;
				吸收液体step:=2;
			END_IF
		2: (* 气隔断: 针尖仍在原位空气中 (5Z=0, XY 未动); 指令为空则跳过 *)
			IF LEN(STR:=Sampling_sample_instructions[2])=0 THEN
				吸收液体step:=8;
			ELSIF %MW1300=0 AND NOT 泵站位符 THEN
				泵站位符:=TRUE;
				转发转存:=Sampling_sample_instructions[2];
				%MW1300:=LEN(STR:=转发转存);
				吸收液体step:=3;
			END_IF
		3: (* 等泵空闲后立即释放总线: 轴移动期间不占共享邮箱 *)
			IF %MW1300=0 AND sample_gap_wait.Q THEN
				转发转存:='/4Q$R';
				%MW1300:=LEN(STR:=转发转存);
			END_IF
			IF sample_gap_idle.Q THEN
				泵站位符:=FALSE;
				吸收液体step:=8;
			END_IF
		8: (* 针尖已成空气段, 此时才移向孔位 *)
			上样轴4X轴DATE.fAbsTarget:=Sampling_4X_Target;
			打样瓶上料轴3YDATE.fAbsTarget:=Sampling_3Y_Target;
			上样轴4X轴DATE.xMoveAbs:=TRUE;
			打样瓶上料轴3YDATE.xMoveAbs:=TRUE;
			吸收液体step:=10;
		10:
			IF 上样轴4X轴DATE.bAbMoveDone AND 打样瓶上料轴3YDATE.bAbMoveDone THEN
				上样轴4X轴DATE.xMoveAbs:=FALSE;
				打样瓶上料轴3YDATE.xMoveAbs:=FALSE;
				上样轴5Z轴DATE.fAbsTarget:=HMI_上样轴5Z轴.position[2];
				上样轴5Z轴DATE.xMoveAbs:=TRUE;
				吸收液体step:=20;
			END_IF
		20: (* 直接解析唯一真源 P<n>，不依赖额外 OPC 伴随参数 *)
			IF 上样轴5Z轴DATE.bAbMoveDone THEN
				上样轴5Z轴DATE.xMoveAbs:=FALSE;
				sample_pB:=ADR(Sampling_sample_instructions[1]);
				sample_relative_steps:=0;
				sample_relative_valid:=FALSE;
				sample_k:=WORD#0;
				WHILE sample_k<=WORD#120 DO
					IF sample_pB[sample_k]=16#50 THEN (* ASCII P *)
						sample_k:=sample_k+WORD#1;
						WHILE (sample_pB[sample_k]>=16#30) AND (sample_pB[sample_k]<=16#39) DO
							sample_relative_steps:=sample_relative_steps*10+(BYTE_TO_INT(sample_pB[sample_k])-48);
							sample_relative_valid:=TRUE;
							sample_k:=sample_k+WORD#1;
						END_WHILE
						EXIT;
					END_IF
					sample_k:=sample_k+WORD#1;
				END_WHILE
				IF sample_relative_valid AND (sample_relative_steps>0) THEN
					sample_q_sent:=FALSE;
					sample_query_retry:=0;
					吸收液体step:=22;
				ELSE
					Sampling_L2_ErrorCode:=463;
					吸收液体step:=90;
				END_IF
			END_IF
		22: (* 获取共享泵总线并查询当前绝对活塞位 *)
			IF %MW1300=0 AND NOT 泵站位符 THEN
				泵站位符:=TRUE;
				接收字符:='';
				转发转存:='/4?$R';
				%MW1300:=LEN(STR:=转发转存);
				sample_q_sent:=TRUE;
				吸收液体step:=23;
			END_IF
		23: (* 解析 /4?；响应不带泵地址，解析完成前不得释放占位 *)
			IF TON[11].Q THEN
				sample_q_sent:=FALSE;
				sample_pB:=ADR(接收字符);
				sample_pos:=0;
				sample_pos_valid:=FALSE;
				sample_k:=WORD#0;
				WHILE sample_k<=WORD#60 DO
					IF (sample_pB[sample_k]=16#2F) AND (sample_pB[sample_k+1]=16#30) THEN
						EXIT;
					END_IF
					sample_k:=sample_k+WORD#1;
				END_WHILE
				IF sample_k<=WORD#60 THEN
					sample_k:=sample_k+WORD#3;
					WHILE (sample_pB[sample_k]>=16#30) AND (sample_pB[sample_k]<=16#39) DO
						sample_pos:=sample_pos*10+(BYTE_TO_INT(sample_pB[sample_k])-48);
						sample_pos_valid:=TRUE;
						sample_k:=sample_k+WORD#1;
					END_WHILE
				END_IF
				IF sample_pos_valid THEN
					IF (sample_relative_steps<=0) OR ((sample_pos+sample_relative_steps)>6000) THEN
						泵站位符:=FALSE;
						Sampling_L2_ErrorCode:=463;
						吸收液体step:=90;
					ELSE
						吸收液体step:=25;
					END_IF
				ELSE
					sample_query_retry:=sample_query_retry+1;
					IF sample_query_retry>5 THEN
						泵站位符:=FALSE;
						Sampling_L2_ErrorCode:=464;
						吸收液体step:=90;
					ELSE
						吸收液体step:=24;
					END_IF
				END_IF
			END_IF
		24: (* 查询无有效帧时，在同一占位内重试 *)
			IF %MW1300=0 AND NOT sample_q_sent THEN
				接收字符:='';
				转发转存:='/4?$R';
				%MW1300:=LEN(STR:=转发转存);
				sample_q_sent:=TRUE;
				吸收液体step:=23;
			END_IF
		25: (* 行程已校验；保持同一总线占位发送 P<n> *)
			IF %MW1300=0 THEN
				转发转存:=Sampling_sample_instructions[1];
				%MW1300:=LEN(STR:=转发转存);
				吸收液体step:=30;
			END_IF
		30:
			IF %MW1300=0 AND TON_0.Q THEN
				转发转存:='/4Q$R';
				%MW1300:=LEN(STR:=转发转存);
			END_IF
			IF R_TRIG[10].Q THEN
				泵站位符:=FALSE;
				吸收液体step:=40;
			END_IF
		40:
			上样轴5Z轴DATE.fAbsTarget:=0;
			上样轴5Z轴DATE.xMoveAbs:=TRUE;
			IF 上样轴5Z轴DATE.bAbMoveDone THEN
				上样轴5Z轴DATE.xMoveAbs:=FALSE;
				Sampling_liquid_absorption:=TRUE;
				吸收液体step:=0;
				bActionDone:=TRUE;
			END_IF
		90: (* 参数/查询错误也先安全抬针再上报 *)
			上样轴5Z轴DATE.fAbsTarget:=0;
			上样轴5Z轴DATE.xMoveAbs:=TRUE;
			IF 上样轴5Z轴DATE.bAbMoveDone THEN
				上样轴5Z轴DATE.xMoveAbs:=FALSE;
				吸收液体step:=0;
				bActionError:=TRUE;
			END_IF
	END_CASE
END_IF
END_ACTION

ACTION A31_放板移轴:
(* 放板移轴: 点样7Y轴到放板位 (上位机随后驱动机器人放板) *)
CASE 放硅胶板STEP OF
	0:
		点样轴7YDATE.fAbsTarget:=HMI_点样轴7Y.position[1];
		点样轴7YDATE.xMoveAbs:=TRUE;
		放硅胶板STEP:=10;
	10:
		IF 点样轴7YDATE.bAbMoveDone THEN
			点样轴7YDATE.xMoveAbs:=FALSE;
			放硅胶板STEP:=0;
			bActionDone:=TRUE;
		END_IF
END_CASE
END_ACTION

ACTION A55_润洗吹打混匀:
(* A55 润洗吹打混匀：回打余量 -> 口1润洗 -> 抬针吸气隔断 -> 下针口3循环吹打 -> 退针 (终态活塞=A{gap}) *)
rinse_mix_wait(
    IN := (rinse_mix_step = 31) OR (rinse_mix_step = 41) OR (rinse_mix_step = 44) OR (rinse_mix_step = 51),
    PT := T#0.5S
);
rinse_mix_idle(CLK := %MX2005.5);

CASE rinse_mix_step OF
    0:
        (* 参数必须在运动前完成防御性校验；四条命令均由上位机翻译, [1][2]以A0结束, [3][4]以A{gap}结束。 *)
        IF (Sampling_rinse_mix_count < 1) OR (Sampling_rinse_mix_count > 20) OR
           (LEN(STR := Sampling_rinse_mix_instructions[1]) = 0) OR
           (LEN(STR := Sampling_rinse_mix_instructions[2]) = 0) OR
           (LEN(STR := Sampling_rinse_mix_instructions[3]) = 0) OR
           (LEN(STR := Sampling_rinse_mix_instructions[4]) = 0) THEN
            上样点样三通电池阀自动 := FALSE;
            Sampling_L2_ErrorCode := 466;
            Sampling_L2_Retryable := FALSE;
            bActionError := TRUE;
        ELSE
            rinse_mix_cycle := 0;
            上样轴5Z轴DATE.fAbsTarget := 0;
            上样轴5Z轴DATE.xMoveAbs := TRUE;
            IF 上样轴5Z轴DATE.bAbMoveDone THEN
                上样轴5Z轴DATE.xMoveAbs := FALSE;
                上样轴4X轴DATE.fAbsTarget := Sampling_4X_Target;
                打样瓶上料轴3YDATE.fAbsTarget := Sampling_3Y_Target;
                上样轴4X轴DATE.xMoveAbs := TRUE;
                打样瓶上料轴3YDATE.xMoveAbs := TRUE;
                rinse_mix_step := 10;
            END_IF
        END_IF

    10:
        IF 上样轴4X轴DATE.bAbMoveDone AND 打样瓶上料轴3YDATE.bAbMoveDone THEN
            上样轴4X轴DATE.xMoveAbs := FALSE;
            打样瓶上料轴3YDATE.xMoveAbs := FALSE;
            上样轴5Z轴DATE.fAbsTarget := HMI_上样轴5Z轴.position[2];
            上样轴5Z轴DATE.xMoveAbs := TRUE;
            rinse_mix_step := 20;
        END_IF

    20:
        IF 上样轴5Z轴DATE.bAbMoveDone THEN
            上样轴5Z轴DATE.xMoveAbs := FALSE;
            (* FALSE 为上样针侧；整个回打/润洗/混匀期间保持在原孔流路。 *)
            上样点样三通电池阀自动 := FALSE;
            rinse_mix_step := 30;
        END_IF

    30: (* 1. 当前活塞内容(上一轮点样驱动液余量)经口3回打到原样品孔，并回 A0 *)
        IF (%MW1300 = 0) AND (NOT 泵站位符) THEN
            泵站位符 := TRUE;
            转发转存 := Sampling_rinse_mix_instructions[1];
            %MW1300 := LEN(STR := 转发转存);
            rinse_mix_step := 31;
        END_IF

    31:
        IF (%MW1300 = 0) AND rinse_mix_wait.Q THEN
            转发转存 := '/4Q$R';
            %MW1300 := LEN(STR := 转发转存);
        END_IF
        IF rinse_mix_idle.Q THEN
            rinse_mix_step := 40;
        END_IF

    40: (* 2. 口1吸润洗液，经口3全部打入原样品孔，并回 A0 *)
        IF %MW1300 = 0 THEN
            转发转存 := Sampling_rinse_mix_instructions[2];
            %MW1300 := LEN(STR := 转发转存);
            rinse_mix_step := 41;
        END_IF

    41:
        IF (%MW1300 = 0) AND rinse_mix_wait.Q THEN
            转发转存 := '/4Q$R';
            %MW1300 := LEN(STR := 转发转存);
        END_IF
        IF rinse_mix_idle.Q THEN
            rinse_mix_cycle := 0;
            rinse_mix_step := 42;
        END_IF

    42: (* 3a. 抬针到0, 针尖离液进入空气, 为吸气隔断做准备 *)
        上样轴5Z轴DATE.fAbsTarget := 0;
        上样轴5Z轴DATE.xMoveAbs := TRUE;
        IF 上样轴5Z轴DATE.bAbMoveDone THEN
            上样轴5Z轴DATE.xMoveAbs := FALSE;
            rinse_mix_step := 43;
        END_IF

    43: (* 3b. 口3吸气隔断至 A{gap}, 隔离混合液与共管清洗液柱 *)
        IF %MW1300 = 0 THEN
            转发转存 := Sampling_rinse_mix_instructions[3];
            %MW1300 := LEN(STR := 转发转存);
            rinse_mix_step := 44;
        END_IF

    44:
        IF (%MW1300 = 0) AND rinse_mix_wait.Q THEN
            转发转存 := '/4Q$R';
            %MW1300 := LEN(STR := 转发转存);
        END_IF
        IF rinse_mix_idle.Q THEN
            rinse_mix_step := 45;
        END_IF

    45: (* 3c. 下针回原孔液面下, 准备带隔断混匀 *)
        上样轴5Z轴DATE.fAbsTarget := HMI_上样轴5Z轴.position[2];
        上样轴5Z轴DATE.xMoveAbs := TRUE;
        IF 上样轴5Z轴DATE.bAbMoveDone THEN
            上样轴5Z轴DATE.xMoveAbs := FALSE;
            rinse_mix_step := 50;
        END_IF

    50: (* 4. 口3吸至A{gap+mix}并打回A{gap}, 按 count 循环吹打, 气隔断全程保留 *)
        IF %MW1300 = 0 THEN
            转发转存 := Sampling_rinse_mix_instructions[4];
            %MW1300 := LEN(STR := 转发转存);
            rinse_mix_step := 51;
        END_IF

    51:
        IF (%MW1300 = 0) AND rinse_mix_wait.Q THEN
            转发转存 := '/4Q$R';
            %MW1300 := LEN(STR := 转发转存);
        END_IF
        IF rinse_mix_idle.Q THEN
            rinse_mix_cycle := rinse_mix_cycle + 1;
            IF rinse_mix_cycle >= Sampling_rinse_mix_count THEN
                泵站位符 := FALSE;
                rinse_mix_step := 60;
            ELSE
                rinse_mix_step := 50;
            END_IF
        END_IF

    60: (* 四条命令均已 Q 空闲确认，泵停在 A{gap}；保持上样侧并安全退针。 *)
        上样点样三通电池阀自动 := FALSE;
        上样轴5Z轴DATE.fAbsTarget := 0;
        上样轴5Z轴DATE.xMoveAbs := TRUE;
        IF 上样轴5Z轴DATE.bAbMoveDone THEN
            上样轴5Z轴DATE.xMoveAbs := FALSE;
            泵站位符 := FALSE;
            rinse_mix_step := 0;
            rinse_mix_cycle := 0;
            bActionDone := TRUE;
        END_IF
END_CASE
END_ACTION

ACTION A40_prep_上样准备:
(* 上样准备: Z回零 -> 从已清洗输出管路绝对回抽驱动清洗液并保留 (仅第1条指令) *)
TON[2](IN:=上样准备step=2, PT:=T#0.5S);
R_TRIG[3](CLK:=%MX2005.5);
CASE 上样准备step OF
	0:
		上样轴5Z轴DATE.fAbsTarget:=0;
		上样轴5Z轴DATE.xMoveAbs:=TRUE;
		IF 上样轴5Z轴DATE.bAbMoveDone THEN
			上样轴5Z轴DATE.xMoveAbs:=FALSE;
			上样准备step:=1;
		END_IF
	1:
		IF %MW1300=0 AND NOT 泵站位符 THEN
			泵站位符:=TRUE;
			转发转存:=Sampling_prep_instructions[1];
			%MW1300:=LEN(STR:=转发转存);
			上样准备step:=2;
		END_IF
	2:
		IF %MW1300=0 AND TON[2].Q THEN
			转发转存:='/4Q$R';
			%MW1300:=LEN(STR:=转发转存);
		END_IF
		IF R_TRIG[3].Q THEN
			泵站位符:=FALSE;
			Sampling_preparation_OK:=TRUE;
			上样准备step:=0;
			bActionDone:=TRUE;
		END_IF
END_CASE
END_ACTION

ACTION A32_放板定位:
(* 放板定位: 上位机放板后定位夹紧 *)
上样定位自动:=TRUE;
Sampling_Place_materials_OK:=TRUE;
bActionDone:=TRUE;
END_ACTION

ACTION A20_clean_清洗:
(* 清洗: 伺服到清洗位 -> 注射泵清洗循环 Sampling_clean_count 次 (纯设备)
   mode=1 轻清洗充液分支 (spec 2026-07-14-sampling-light-flush §3.3): 步 110-140,
   entry[1]=吸满+充上样流路+冲外壁(链式, 阀FALSE=上样针侧), entry[2]=冲点样头至A0(阀TRUE=点样头侧);
   切阀恒在 entry 边界且 /4Q 确认泵空闲后; 完成复位阀到上样针侧; 不进 Sampling_clean_count 循环。
   Sampling_clean_mode 由上位机每次派发显式写 (0=重清洗现行/1=轻清洗), PLC 只读不复位。 *)
TON[1](IN:=清洗step=20,PT:=T#0.5S);
TON[6](IN:=清洗step=40,PT:=T#0.5S);
TON[8](IN:=清洗step=26,PT:=T#0.5S);
TON[3](IN:=清洗step=120,PT:=T#0.5S);
TON[9](IN:=清洗step=140,PT:=T#0.5S);
R_TRIG[2](CLK:=%MX2005.5);
R_TRIG[11](CLK:=%MX2005.5);
R_TRIG[12](CLK:=%MX2005.5);
R_TRIG[4](CLK:=%MX2005.5);
R_TRIG[5](CLK:=%MX2005.5);
CASE 清洗step OF
	0 :
		点样轴6XDATE.xMoveAbs:=FALSE;
		上样轴4X轴DATE.xMoveAbs:=FALSE;
		上样轴5Z轴DATE.xMoveAbs:=FALSE;
		清洗step:=2;
	
	2:
		上样轴5Z轴DATE.fAbsTarget:=0;
		上样轴5Z轴DATE.xMoveAbs:=TRUE;
		IF 上样轴5Z轴DATE.bAbMoveDone THEN
			上样轴5Z轴DATE.xMoveAbs:=FALSE;
			清洗step:=5;
		END_IF
	5:
		点样轴6XDATE.fAbsTarget:=HMI_点样轴6X.position[1];
// 		上样轴4X轴DATE.fAbsTarget:=HMI_上样轴4X轴.position[9];
		上样轴4X轴DATE.fAbsTarget:=Sampling_4X_WashTarget;
		点样轴6XDATE.xMoveAbs:=TRUE;
		上样轴4X轴DATE.xMoveAbs:=TRUE;
		清洗计数:=0;
		清洗step:=6;
	6:
		IF 上样轴4X轴DATE.bAbMoveDone THEN
			上样轴4X轴DATE.xMoveAbs:=FALSE;
			上样轴5Z轴DATE.fAbsTarget:=HMI_上样轴5Z轴.position[1];
			上样轴5Z轴DATE.xMoveAbs:=TRUE;
			清洗step:=7;
		END_IF
	7:
		IF  上样轴5Z轴DATE.bAbMoveDone AND 点样轴6XDATE.bAbMoveDone THEN
			上样轴5Z轴DATE.xMoveAbs:=FALSE;
			点样轴6XDATE.xMoveAbs:=FALSE;
			IF Sampling_clean_mode=1 THEN
				清洗step:=110;
			ELSIF Sampling_clean_count>0 THEN
				清洗step:=10;
			ELSE
				清洗step:=60;
			END_IF
		END_IF
	10:
		IF %MW1300=0 AND NOT 泵站位符 THEN
			泵站位符:=TRUE;
			转发转存:=Sampling_clean_instructions[1];
			%MW1300:=LEN(STR:= 转发转存);
			上样点样三通电池阀自动:=TRUE;
			清洗step:=20;
		END_IF
	20:
		IF %MW1300=0 AND TON[1].Q THEN
		转发转存:='/4Q$R';
		%MW1300:=LEN(STR:= 转发转存);
		END_IF
		IF R_TRIG[2].Q THEN
			上样点样三通电池阀自动:=FALSE;
			泵站位符:=FALSE;
			清洗step:=24;
		END_IF
	24:
		IF %MW1300=0 AND NOT 泵站位符 THEN
			泵站位符:=TRUE;
			转发转存:=Sampling_clean_instructions[1];
			%MW1300:=LEN(STR:= 转发转存);
			清洗step:=26;
		END_IF
	26:
		IF %MW1300=0 AND TON[8].Q THEN
		转发转存:='/4Q$R';
		%MW1300:=LEN(STR:= 转发转存);
		END_IF
		IF R_TRIG[11].Q THEN
			泵站位符:=FALSE;
			清洗step:=30;
		END_IF
	30:
		IF %MW1300=0 AND NOT 泵站位符 THEN
			泵站位符:=TRUE;
			转发转存:=Sampling_clean_instructions[2];
			%MW1300:=LEN(STR:= 转发转存);
			清洗step:=40;
		END_IF
	40:
		IF %MW1300=0 AND TON[6].Q THEN
		转发转存:='/4Q$R';
		%MW1300:=LEN(STR:= 转发转存);
		END_IF
		IF R_TRIG[12].Q THEN
			泵站位符:=FALSE;
			清洗step:=50;
		END_IF
	50:
		清洗计数:=清洗计数+1;
		IF  Sampling_clean_count> 清洗计数 THEN
			转发转存:='';
			%MW1300:=128;
			清洗step:=10;
		ELSIF  Sampling_clean_count<= 清洗计数 THEN
			转发转存:='';
			%MW1300:=128;
			清洗计数:=0;
			Sampling_Cleaning_OK:=TRUE;
			清洗step:=0;
			bActionDone:=TRUE;
		END_IF
		上样点样三通电池阀自动:=FALSE;
	60:
		Sampling_Cleaning_OK:=TRUE;
		清洗step:=0;
		bActionDone:=TRUE;
	(* ===== mode=1 轻清洗充液 (spec 2026-07-14-sampling-light-flush) ===== *)
	110: (* 派发 entry[1]: 吸满+充上样流路+冲外壁; 三通=上样针侧(FALSE) *)
		IF %MW1300=0 AND NOT 泵站位符 THEN
			泵站位符:=TRUE;
			转发转存:=Sampling_clean_instructions[1];
			%MW1300:=LEN(STR:= 转发转存);
			上样点样三通电池阀自动:=FALSE;
			清洗step:=120;
		END_IF
	120: (* /4Q 确认泵空闲 -> 切三通到点样头侧(TRUE) *)
		IF %MW1300=0 AND TON[3].Q THEN
		转发转存:='/4Q$R';
		%MW1300:=LEN(STR:= 转发转存);
		END_IF
		IF R_TRIG[4].Q THEN
			泵站位符:=FALSE;
			上样点样三通电池阀自动:=TRUE;
			清洗step:=130;
		END_IF
	130: (* 派发 entry[2]: 冲点样头至 A0; 三通保持点样头侧 *)
		IF %MW1300=0 AND NOT 泵站位符 THEN
			泵站位符:=TRUE;
			转发转存:=Sampling_clean_instructions[2];
			%MW1300:=LEN(STR:= 转发转存);
			清洗step:=140;
		END_IF
	140: (* /4Q 确认泵空闲 -> 复位三通到上样针侧, 完成 *)
		IF %MW1300=0 AND TON[9].Q THEN
		转发转存:='/4Q$R';
		%MW1300:=LEN(STR:= 转发转存);
		END_IF
		IF R_TRIG[5].Q THEN
			泵站位符:=FALSE;
			上样点样三通电池阀自动:=FALSE;
			Sampling_Cleaning_OK:=TRUE;
			清洗step:=0;
			bActionDone:=TRUE;
		END_IF
END_CASE
END_ACTION

ACTION A62_单条带点样:
(* A62 单条带点样 — 模型B ③(E+B): 蛇形双向液体程 + 到位即停泵起吹干(去驻留), /4? 查询并行化
   spec: 2026-07-14-band-edge-artifacts v3 §3 + 2026-07-14-spot-end-position §3.5
//    每程: A{N}R 供液 -> 按 dir 扫线到位 -> 发T即起吹干leg1(反向离开停点), /4?+沉降200ms+解析并行块
   -> dry_cycles 周期(每周期2 leg, 终点=本程停点) -> step38 判终: pos<=Sampling_band_end_position+5
   收尾, 否则 dir 取反从当前端直发下一程 (旧回程 step40/42 已删)。
   死锁纪律不变: xMoveAbs 置位步与 done 原子消费步一一配对; 泵站位符 发A{N}R起持有至 /4? 有效响应。
   保险: 单带最多60程(462); 查询无效重试5次(465: 停轴+关气关阀+恢复速度, 跳惰性步99等父接管,
   不得直设 step0 — 并行块在 CASE 前, 同周期会被 step0 的回程命令穿透撤销急停)。 *)
TON[10](IN := spot_band_q_sent, PT := T#200MS);
Sampling_L2_Step := spot_band_step;

(* —— /4? 并行查询块: 与轴运动同周期跑; 泵站位符 在此释放 —— *)
IF spot_band_query_active THEN
	IF %MW1300 = 0 AND NOT spot_band_q_sent THEN
		接收字符 := '';
		转发转存 := '/4?$R';
		%MW1300 := LEN(STR:=转发转存);
		spot_band_q_sent := TRUE;
	END_IF
	IF TON[10].Q THEN
		spot_band_q_sent := FALSE;
		spot_band_pB := ADR(接收字符);
		spot_band_pos := 0;
		spot_band_pos_valid := FALSE;
		spot_band_k := 0;
		WHILE spot_band_k <= 60 DO
			IF (spot_band_pB[spot_band_k] = 16#2F) AND (spot_band_pB[spot_band_k + 1] = 16#30) THEN
				EXIT;
			END_IF
			spot_band_k := spot_band_k + 1;
		END_WHILE
		IF spot_band_k <= 60 THEN
			spot_band_k := spot_band_k + 3;
			WHILE (spot_band_pB[spot_band_k] >= 16#30) AND (spot_band_pB[spot_band_k] <= 16#39) DO
				spot_band_pos := spot_band_pos * 10 + (BYTE_TO_INT(spot_band_pB[spot_band_k]) - 48);
				spot_band_pos_valid := TRUE;
				spot_band_k := spot_band_k + 1;
			END_WHILE
		END_IF
		IF spot_band_pos_valid THEN
			(* /4? 有效响应已完整归属本事务，此时才允许释放共享泵总线。 *)
			泵站位符 := FALSE;
			spot_band_query_retry := 0;
			spot_band_query_active := FALSE;
			spot_band_query_done := TRUE;
		ELSE
			(* 无效/未完整响应不能当作"未到目标"；保持占位并重查。 *)
			spot_band_query_retry := spot_band_query_retry + 1;
			IF spot_band_query_retry > 5 THEN
				泵站位符 := FALSE;
				spot_band_query_active := FALSE;
				点样轴6XDATE.xMoveAbs := FALSE;   (* 轴可能在吹干 leg 中: 立即停轴 *)
				上样吹气自动 := FALSE;
				上样点样三通电池阀自动 := FALSE;
				IF spot_band_velocity_saved THEN
					点样轴6XDATE.fVelocity := spot_band_old_6x_velocity;
					spot_band_velocity_saved := FALSE;
				END_IF
				Sampling_L2_ErrorCode := 465;
				spot_band_step := 99;
				bActionError := TRUE;
			END_IF
		END_IF
	END_IF
END_IF

CASE spot_band_step OF
	0:
		IF NOT spot_band_velocity_saved THEN
			spot_band_old_6x_velocity := 点样轴6XDATE.fVelocity;
			spot_band_velocity_saved := TRUE;
		END_IF
		IF Sampling_band_dry_cycles < 1 THEN
			Sampling_band_dry_cycles := 1;
		END_IF
		点样轴6XDATE.xMoveAbs := FALSE;
		点样轴7YDATE.xMoveAbs := FALSE;
		上样点样三通电池阀自动 := FALSE;
		上样吹气自动 := FALSE;
		泵站位符 := FALSE;   (* 防御性释放: 上次运行非常规中断残留 TRUE 会使 step12 静默死锁 *)
		spot_band_q_sent := FALSE;
		spot_band_pass_count := 0;
		spot_band_query_retry := 0;
		spot_band_dir := TRUE;
		spot_band_query_active := FALSE;
		spot_band_query_done := FALSE;
		IF Sampling_band_spot_speed > 0.0 THEN
			点样轴6XDATE.fVelocity := Sampling_band_spot_speed;
		END_IF
		点样轴6XDATE.fAbsTarget := Spot_6X_StartTarget;
		点样轴7YDATE.fAbsTarget := Spot_7Y_Target;
		点样轴6XDATE.xMoveAbs := TRUE;
		点样轴7YDATE.xMoveAbs := TRUE;
		spot_band_step := 10;
	10: (* 到起点(原子消费两轴 done); 第1程恒正向 *)
		IF 点样轴6XDATE.bAbMoveDone AND 点样轴7YDATE.bAbMoveDone THEN
			点样轴6XDATE.xMoveAbs := FALSE;
			点样轴7YDATE.xMoveAbs := FALSE;
			spot_band_step := 12;
		END_IF
	12: (* 发一程供液 A{N}R (泵朝目标N), 阀->点样头, 气ON; 程数保险; 蛇形下头已在本程起点 *)
		IF %MW1300 = 0 AND NOT 泵站位符 THEN
			spot_band_pass_count := spot_band_pass_count + 1;
			IF spot_band_pass_count > 60 THEN
				Sampling_L2_ErrorCode := 462;
				bActionError := TRUE;
				spot_band_step := 0;
			ELSE
				上样点样三通电池阀自动 := TRUE;
				上样吹气自动 := TRUE;
				泵站位符 := TRUE;
				spot_band_query_done := FALSE;
				转发转存 := Sampling_band_run_instruction;
				%MW1300 := LEN(STR:=转发转存);
				spot_band_step := 15;
			END_IF
		END_IF
	15: (* A{N}R 已送出 -> 按 dir 起本程扫线 (点样速) *)
		IF %MW1300 = 0 THEN
			IF Sampling_band_spot_speed > 0.0 THEN
				点样轴6XDATE.fVelocity := Sampling_band_spot_speed;
			END_IF
			IF spot_band_dir THEN
				点样轴6XDATE.fAbsTarget := Spot_6X_EndTarget;
			ELSE
				点样轴6XDATE.fAbsTarget := Spot_6X_StartTarget;
			END_IF
			点样轴6XDATE.xMoveAbs := TRUE;
			spot_band_step := 20;
		END_IF
	20: (* 扫线到位 【唯一写者/唯一消费】 *)
		上样点样三通电池阀自动 := TRUE;
		上样吹气自动 := TRUE;
		IF 点样轴6XDATE.bAbMoveDone THEN
			点样轴6XDATE.xMoveAbs := FALSE;
			spot_band_q_sent := FALSE;
			spot_band_query_retry := 0;
			spot_band_step := 24;
		END_IF
	24: (* E核心: 停泵 /4T -> 启动并行查询, 立即转吹干(不在停点驻留) *)
		上样点样三通电池阀自动 := TRUE;
		上样吹气自动 := TRUE;
		IF %MW1300 = 0 THEN
			转发转存 := '/4T$R';
			%MW1300 := LEN(STR:=转发转存);
			spot_band_query_active := TRUE;
			spot_band_dry_count := 0;
			spot_band_step := 30;
		END_IF
	30: (* 吹干 leg1: 反向离开本程停点 (吹干速); T送达前后余液被运动摊开 *)
		上样点样三通电池阀自动 := TRUE;
		上样吹气自动 := TRUE;
		IF Sampling_band_dry_speed > 0.0 THEN
			点样轴6XDATE.fVelocity := Sampling_band_dry_speed;
		END_IF
		IF spot_band_dir THEN
			点样轴6XDATE.fAbsTarget := Spot_6X_StartTarget;
		ELSE
			点样轴6XDATE.fAbsTarget := Spot_6X_EndTarget;
		END_IF
		点样轴6XDATE.xMoveAbs := TRUE;
		spot_band_step := 32;
	32:
		IF 点样轴6XDATE.bAbMoveDone THEN
			点样轴6XDATE.xMoveAbs := FALSE;
			spot_band_step := 34;
		END_IF
	34: (* 吹干 leg2: 回本程停点 (= 蛇形下一程起点) *)
		上样点样三通电池阀自动 := TRUE;
		上样吹气自动 := TRUE;
		IF Sampling_band_dry_speed > 0.0 THEN
			点样轴6XDATE.fVelocity := Sampling_band_dry_speed;
		END_IF
		IF spot_band_dir THEN
			点样轴6XDATE.fAbsTarget := Spot_6X_EndTarget;
		ELSE
			点样轴6XDATE.fAbsTarget := Spot_6X_StartTarget;
		END_IF
		点样轴6XDATE.xMoveAbs := TRUE;
		spot_band_step := 36;
	36:
		IF 点样轴6XDATE.bAbMoveDone THEN
			点样轴6XDATE.xMoveAbs := FALSE;
			spot_band_dry_count := spot_band_dry_count + 1;
			IF spot_band_dry_count >= Sampling_band_dry_cycles THEN
				spot_band_step := 38;
			ELSE
				spot_band_step := 30;
			END_IF
		END_IF
	38: (* 判终等待: 头已停回本程停点, 等并行查询解析 (正常吹干时长>>查询, 不驻留) *)
		上样点样三通电池阀自动 := TRUE;
		上样吹气自动 := TRUE;
		IF spot_band_query_done THEN
			spot_band_query_done := FALSE;
			IF spot_band_pos <= Sampling_band_end_position + 5 THEN
				spot_band_step := 70;
			ELSE
				spot_band_dir := NOT spot_band_dir;
				spot_band_step := 12;
			END_IF
		END_IF
	70: (* 收尾: 带气到清洗位 -> 关气 -> 复位 (蛇形下起点可为 Start/End 侧, X包络为基线已扫范围子集) *)
		上样点样三通电池阀自动 := TRUE;
		上样吹气自动 := TRUE;
		点样轴6XDATE.fAbsTarget := HMI_点样轴6X.position[1];
		点样轴6XDATE.xMoveAbs := TRUE;
		spot_band_step := 80;
	80:
		IF 点样轴6XDATE.bAbMoveDone THEN
			点样轴6XDATE.xMoveAbs := FALSE;
			点样轴7YDATE.fAbsTarget := HMI_点样轴7Y.position[1];
			点样轴7YDATE.xMoveAbs := TRUE;
			spot_band_step := 90;
		END_IF
	90:
		IF 点样轴7YDATE.bAbMoveDone THEN
			点样轴7YDATE.xMoveAbs := FALSE;
			上样吹气自动 := FALSE;
			上样点样三通电池阀自动 := FALSE;
			IF spot_band_velocity_saved THEN
				点样轴6XDATE.fVelocity := spot_band_old_6x_velocity;
				spot_band_velocity_saved := FALSE;
			END_IF
			Sampling_Spray_sample_OK := TRUE;
			spot_band_step := 0;
			bActionDone := TRUE;
		END_IF
	99: (* 465 错误保持: 惰性等待父派发器接管终态/Reset, 不发任何运动/输出 *)
		;
END_CASE
END_ACTION

ACTION A10_init_初始化:
(* 初始化: 复位阀/伺服回零 + 注射泵初始化 (已删机器人握手位复位) *)
CASE 初始化step OF
	0 :
		上样定位手动:=FALSE;
		上样定位自动:=FALSE;
		上样点样三通电池阀手动:=FALSE;
		上样点样三通电池阀自动:=FALSE;
		上样吹气手动:=FALSE;
		上样吹气自动:=FALSE;
		打样瓶上料轴3YDATE.fAbsTarget:=0;
		点样轴6XDATE.fAbsTarget:=0;
		点样轴7YDATE.fAbsTarget:=0;
		上样轴4X轴DATE.fAbsTarget:=0;
		上样轴5Z轴DATE.fAbsTarget:=0;
		点样轴7YDATE.xMoveAbs:=FALSE;
		点样轴6XDATE.xMoveAbs:=FALSE;
		上样轴5Z轴DATE.xMoveAbs:=FALSE;
		上样轴4X轴DATE.xMoveAbs:=FALSE;
		打样瓶上料轴3YDATE.xMoveAbs:=FALSE;
		Sampling_Spray_sample_OK:=FALSE;
		Sampling_liquid_absorption:=FALSE;
		Sampling_preparation_OK:=FALSE;
		大真空泵站位[11]:=FALSE;
		清洗计数:=0;
		清洗step:=0;
		放硅胶板STEP:=0;
		上样准备step:=0;
		吸收液体step:=0;
		点样step:=0;
		初始化step:=5;
	5:
		上样轴5Z轴DATE.fAbsTarget:=0;
		上样轴5Z轴DATE.xMoveAbs:=TRUE;
		IF 上样轴5Z轴DATE.bAbMoveDone THEN
			点样轴7YDATE.fAbsTarget:=0  ;
			点样轴6XDATE.fAbsTarget:=0  ;
			上样轴4X轴DATE.fAbsTarget:=0;
			上样轴4X轴DATE.xMoveAbs:=TRUE;
			点样轴7YDATE.xMoveAbs:=TRUE;
			点样轴6XDATE.xMoveAbs:=TRUE;
			初始化step:=6;
		END_IF
	6:
		IF 上样轴4X轴DATE.bAbMoveDone AND 上样轴5Z轴DATE.bAbMoveDone AND 点样轴6XDATE.bAbMoveDone AND 点样轴7YDATE.bAbMoveDone THEN
			初始化step:=10;
			上样轴4X轴DATE.xMoveAbs:=FALSE;
			点样轴7YDATE.xMoveAbs:=FALSE;
			上样轴5Z轴DATE.xMoveAbs:=FALSE;
			点样轴6XDATE.xMoveAbs:=FALSE;
		END_IF
	10:
		IF %MW1300=0 AND NOT 泵站位符 THEN
			泵站位符:=TRUE;
			转发转存:='/4Z0,1,1R$R';
			%MW1300:=LEN(STR:= 转发转存);
			初始化STEP:=20;
		END_IF
	20:
		IF %MW1300=0 THEN
			转发转存:='/4Q$R';
			%MW1300:=LEN(STR:= 转发转存);
		END_IF
		R_TRIG[1](CLK:=%MX2005.5);
		IF R_TRIG[1].Q THEN
			泵站位符:=FALSE;
			初始化STEP:=30;
		END_IF
	30:
		Sampling_initialization_OK:=TRUE;
		初始化step:=0;
		bActionDone:=TRUE;
END_CASE
END_ACTION

ACTION A60_spray_点样:
(* 点样: 伺服点样序列 + 注射泵点样 (已删尾部 允许取硅胶板 机器人握手) *)
TON[4](IN:=点样step=20,PT:=T#0.5S);
TON[5](IN:=点样气泡传感器,PT:=T#5S);
TON[7](IN:=点样step=10,PT:=T#0.5S);
R_TRIG[10](CLK:=%MX2005.5);
CASE 点样step OF
	0:
		点样轴6XDATE.xMoveAbs:=FALSE;
		点样轴7YDATE.xMoveAbs:=FALSE;
		点样step:=1;
	1:
// 		点样轴6XDATE.fAbsTarget:=HMI_点样轴6X.position[2];
		点样轴6XDATE.fAbsTarget:=Spot_6X_StartTarget;
// 		点样轴7YDATE.fAbsTarget:=HMI_点样轴7Y.position[2];
		点样轴7YDATE.fAbsTarget:=Spot_7Y_Target;
		点样轴6XDATE.xMoveAbs:=TRUE;
		点样轴7YDATE.xMoveAbs:=TRUE;
		点样step:=5;
	5:
		IF 点样轴6XDATE.bAbMoveDone AND 点样轴7YDATE.bAbMoveDone THEN
			点样轴6XDATE.xMoveAbs:=FALSE;
			点样轴7YDATE.xMoveAbs:=FALSE;
			IF  %MW1300=0 AND NOT 泵站位符 THEN
				泵站位符:=TRUE;
				转发转存:=Sampling_dispense_instructions[1];
				%MW1300:=LEN(STR:= 转发转存);
				上样点样三通电池阀自动:=TRUE;
				点样step:=10;
			END_IF
		END_IF
	10:
		IF  %MW1300=0 AND TON[7].Q THEN
				转发转存:='/4Q$R';
				%MW1300:=LEN(STR:= 转发转存);
				IF R_TRIG[10].Q THEN
					泵站位符:=FALSE;
					点样step:=15;
				END_IF
		END_IF
	15:
		IF  %MW1300=0 AND NOT 泵站位符 THEN
			上样吹气自动:=TRUE;
			泵站位符:=TRUE;
			转发转存:=Sampling_dispense_instructions[2];
			%MW1300:=LEN(STR:= 转发转存);
// 			点样轴6XDATE.fAbsTarget:=HMI_点样轴6X.position[3];
			点样轴6XDATE.fAbsTarget:=Spot_6X_EndTarget;
			点样轴6XDATE.xMoveAbs:=TRUE;
			点样step:=20;
		END_IF
	20:
		IF  %MW1300=0 AND TON[4].Q THEN
				转发转存:='/4Q$R';
				%MW1300:=LEN(STR:= 转发转存);
				IF R_TRIG[10].Q THEN
					泵站位符:=FALSE;
					上样点样三通电池阀自动:=FALSE;
					上样吹气自动:=FALSE;
				END_IF
		END_IF
		CASE 打样伺服移动step OF
			0:
				IF 点样轴6XDATE.bAbMoveDone THEN
					点样轴6XDATE.xMoveAbs:=FALSE;
					IF 泵站位符 THEN
						打样伺服移动step:=10;
					ELSE
						点样step:=30;
					END_IF
				END_IF
			10:
// 				点样轴6XDATE.fAbsTarget:=HMI_点样轴6X.position[2];
				点样轴6XDATE.fAbsTarget:=Spot_6X_StartTarget;
				点样轴6XDATE.xMoveAbs:=TRUE;
				打样伺服移动step:=20;
			20:
				IF 点样轴6XDATE.bAbMoveDone THEN
					点样轴6XDATE.xMoveAbs:=FALSE;
					打样伺服移动step:=30;
				END_IF
			30:
// 				点样轴6XDATE.fAbsTarget:=HMI_点样轴6X.position[3];
				点样轴6XDATE.fAbsTarget:=Spot_6X_EndTarget;
				点样轴6XDATE.xMoveAbs:=TRUE;
				打样伺服移动step:=0;
		END_CASE
	30:
		点样轴6XDATE.fAbsTarget:=HMI_点样轴6X.position[1];
		点样轴6XDATE.xMoveAbs:=TRUE;
		IF 点样轴6XDATE.bAbMoveDone THEN
			点样轴7YDATE.fAbsTarget:=HMI_点样轴7Y.position[1];
			点样轴7YDATE.xMoveAbs:=TRUE;
			点样step:=40;
		END_IF
	40:
		IF 点样轴7YDATE.bAbMoveDone  THEN
			点样轴6XDATE.xMoveAbs:=FALSE;
			点样轴7YDATE.xMoveAbs:=FALSE;
			上样定位自动:=FALSE;
			Sampling_Spray_sample_OK:=TRUE;
			点样step:=0;
			bActionDone:=TRUE;
		END_IF
END_CASE
END_ACTION

ACTION A61_喷涂移轴:
CASE 喷涂移轴step OF
					0:
						点样轴7YDATE.fAbsTarget := HMI_点样轴7Y.position[2];
						点样轴7YDATE.xMoveAbs := TRUE;
						喷涂移轴step := 10;
					10:
						IF 点样轴7YDATE.bAbMoveDone THEN
							点样轴7YDATE.xMoveAbs := FALSE;
							喷涂移轴step := 0;
							bActionDone := TRUE;
						END_IF
				END_CASE
END_ACTION

END_PROGRAM

// Device/Application/50_action/Collect_L2
PROGRAM Collect_L2
VAR
	初始化STEP: INT;
	准备step: INT;
	收集step: INT;
	搬运step: INT;
	泵初始化完成: BOOL;
	bActionDone: BOOL;
	bActionError: BOOL;
	L2_StartTrig: R_TRIG;
	R_TRIG: ARRAY[1..5] OF R_TRIG;
	ton: ARRAY[1..10] OF TON;
	TON_0: TON;
END_VAR

(* 收集工位 L2 统一动作派发器
   功能:
       按 Collect_L2_ActionCode 把上位机请求派发到设备原子动作 (纯设备, 不含机器人握手).
   协议:
       Collect_L2_Start 上升沿接受请求 -> RUNNING 每周期调用对应原子 -> 原子置 bActionDone -> DONE.
   动作码:
       10 init 初始化 / 21 夹持夹紧 / 22 伸缩伸出 / 23 缩回升降下压
       30 collect 收集 / 41 复位伸出 / 42 伸缩缩回 / 43 松夹持
   参数:
       无, 经 Collect_L2_* 反馈. *)
L2_StartTrig(CLK := Collect_L2_Start);

(* Global deployment/startup gate: reject before any physical action is dispatched. *)
IF L2_StartTrig.Q AND (Collect_L2_State=0)
	AND ((NOT PLC_Ready) OR (PLC_Deploy_State<>0)) THEN
	Collect_L2_AcceptedSeq := Collect_L2_RequestSeq;
	Collect_L2_ActiveCode := Collect_L2_ActionCode;
	Collect_L2_ErrorCode := 190;
	Collect_L2_Retryable := TRUE;
	Collect_L2_CompletedSeq := Collect_L2_RequestSeq;
	Collect_L2_State := 30;
	RETURN;
END_IF

CASE Collect_L2_State OF
	0:  (* IDLE *)
		Collect_L2_Step := 0;
		IF L2_StartTrig.Q THEN
			Collect_L2_AcceptedSeq := Collect_L2_RequestSeq;
			Collect_L2_ActiveCode  := Collect_L2_ActionCode;
			Collect_L2_ErrorCode   := 0;
			Collect_L2_Retryable   := FALSE;
			bActionDone            := FALSE;
			bActionError           := FALSE;
			初始化STEP := 0;
			准备step   := 0;
			收集step   := 0;
			搬运step   := 0;
			CASE Collect_L2_ActionCode OF
				10, 21, 22, 23, 24, 30, 41, 42, 43:
					Collect_L2_SafeState := 0;
					Collect_L2_State     := 10;   (* RUNNING *)
			ELSE
				Collect_L2_ErrorCode    := 101;  (* 未知动作码 *)
				Collect_L2_Retryable    := TRUE;
				Collect_L2_CompletedSeq := Collect_L2_AcceptedSeq;
				Collect_L2_State        := 30;   (* REJECTED *)
			END_CASE
		END_IF

	10: (* RUNNING *)
		IF Collect_L2_Reset THEN Collect_L2_State := 0; RETURN; END_IF   (* RUNNING 中 RESET: 中止挂死动作 *)
		CASE Collect_L2_ActiveCode OF
			10: A10_init_初始化();
			21: A21_夹持夹紧();
			22: A22_伸缩伸出();
			23: A23_缩回升降下压();
			24: 溶液收集瓶定位自动:=Collect_BottleLocate_Target; bActionDone:=TRUE;
			30: A30_collect_收集();
			41: A41_复位伸出();
			42: A42_伸缩缩回();
			43: A43_松夹持();
		END_CASE
		IF bActionDone THEN
			bActionDone             := FALSE;
			Collect_L2_CompletedSeq := Collect_L2_AcceptedSeq;
			Collect_L2_State        := 20;   (* DONE *)
		ELSIF bActionError THEN              (* 设备预条件未满足 -> 报错交上位机 *)
			bActionError            := FALSE;
			Collect_L2_Retryable    := TRUE;
			Collect_L2_CompletedSeq := Collect_L2_AcceptedSeq;
			Collect_L2_State        := 40;   (* ERROR; ErrorCode 由原子置 *)
		END_IF

	20, 30, 40, 50:  (* 终态: 等 Start 落沿或 Reset 回 IDLE *)
		IF (NOT Collect_L2_Start) OR Collect_L2_Reset THEN
			Collect_L2_State := 0;
		END_IF
END_CASE

ACTION A23_缩回升降下压:
(* 缩回 -> 升降上升 -> 下压 (上位机已先驱动机器人放收集瓶)
   缺瓶处理: 原 A10 "缺瓶重试" 改为报错交上位机 (ErrorCode 201), 由上位机重放瓶后重调 *)
CASE 准备step OF
	0:
		收集伸缩气缸自动:=FALSE;
		准备step:=10;
	10:
		IF 收集平台推出气缸原点 AND 收集平台瓶子有无传感器 THEN
			收集升降气缸自动:=TRUE;
			准备step:=20;
		ELSIF 收集平台推出气缸原点 AND NOT 收集平台瓶子有无传感器 THEN
			准备step:=0;
			Collect_L2_ErrorCode:=201;   (* 缺瓶: 上位机放瓶后传感器未检到 *)
			bActionError:=TRUE;
		END_IF
	20:
		IF 收集平台升降气缸动点 THEN
			收集下压气缸自动:=TRUE;
			准备step:=0;
			bActionDone:=TRUE;
		END_IF
END_CASE
END_ACTION

ACTION A22_伸缩伸出:
(* 伸缩气缸伸出到放瓶位 *)
CASE 准备step OF
	0:
		IF 收集平台推出气缸原点 AND NOT 收集平台瓶子有无传感器 THEN
			收集伸缩气缸自动:=TRUE;
			准备step:=10;
		END_IF
	10:
		IF 收集平台推出气缸动点 THEN
			准备step:=0;
			bActionDone:=TRUE;
		END_IF
END_CASE
END_ACTION

ACTION A21_夹持夹紧:
(* 夹持气缸夹紧 (上位机已先驱动机器人放收集器) *)
CASE 准备step OF
	0:
		收集夹持气缸自动:=TRUE;
		准备step:=10;
	10:
		IF 收集平台夹持气缸动点 THEN
			准备step:=0;
			bActionDone:=TRUE;
		END_IF
END_CASE
END_ACTION

ACTION A30_collect_收集:
(* 收集: 进液 -> 注射泵转发 -> 排液/正压循环 collect_count 次 (纯设备, 不变) *)
ton[1](IN:=收集step=10, PT:=T#0.5S);
ton[2](IN:=收集step=30, PT:=T#20S);
R_TRIG[5](CLK := %MX2005.5);
CASE 收集step OF
	0:
		IF collect_forward_instructions<>'' THEN
			收集进液自动:=TRUE;
		END_IF
		IF %MW1300=0 AND 泵站位符=FALSE THEN
			转发转存:=collect_forward_instructions;
			%MW1300:=LEN(STR:= 转发转存);
			泵站位符:=TRUE;
			收集step:=10;
		END_IF
	10:
		IF %MW1300=0 AND ton[1].Q THEN
			转发转存:='/3Q$R';
			%MW1300:=LEN(STR:= 转发转存);
		END_IF
		IF R_TRIG[5].Q THEN
			泵站位符:=FALSE;
			收集step:=20;
		END_IF
	20:
		转发转存:='';
		%MW1300:=128;
		收集进液自动:=FALSE;
		收集排液自动:=TRUE;
		收集正压排液自动:=TRUE;
		收集计数:=收集计数+1;
		收集step:=30;
	30:
		TON_0(IN:=ton[2].Q, PT:=T#5S);   (* 排液计时后再沉淀, 沉淀完成才判定, 杜绝误回 step0 *)
		IF TON_0.Q THEN
			IF 收集计数>=collect_count THEN
				收集计数:=0;
				收集step:=40;
			ELSE
				收集排液自动:=FALSE;
				收集正压排液自动:=FALSE;
				收集step:=0;
			END_IF
		END_IF
	40:
		收集排液自动:=FALSE;
		收集正压排液自动:=FALSE;
		收集step:=0;
		bActionDone:=TRUE;
END_CASE
END_ACTION

ACTION A10_init_初始化:
(* 初始化: 复位气缸/电磁阀 + 注射泵初始化 (已删机器人握手位复位)
   完成条件: 四气缸回原点 AND 泵初始化完成 *)
R_TRIG[1](CLK := %MX2005.5);   (* 泵空闲上升沿 *)
CASE 初始化STEP OF
	0:
		溶液收集瓶定位自动:=FALSE;
		收集下压气缸手动:=FALSE; 收集下压气缸自动:=FALSE;
		收集夹持气缸手动:=FALSE; 收集夹持气缸自动:=FALSE;
		收集升降气缸手动:=FALSE; 收集升降气缸自动:=FALSE;
		收集伸缩气缸手动:=FALSE; 收集伸缩气缸自动:=FALSE;
		收集进液手动:=FALSE; 收集进液自动:=FALSE;
		收集排液手动:=FALSE; 收集排液自动:=FALSE;
		收集正压排液手动:=FALSE; 收集正压排液自动:=FALSE;
		溶液收集瓶定位手动:=FALSE;
		IF %MW1300=0 AND NOT 泵站位符 THEN
			泵站位符:=TRUE;
			转发转存:='/3Z0,2,2R$R';             (* 泵初始化指令 *)
			%MW1300:=LEN(STR:= 转发转存);
			初始化STEP:=10;
		END_IF
	10:
		IF %MW1300=0 THEN
			转发转存:='/3Q$R';                   (* 查询泵状态 *)
			%MW1300:=LEN(STR:= 转发转存);
		END_IF
		IF R_TRIG[1].Q THEN
			泵站位符:=FALSE;
			泵初始化完成:=TRUE;
			初始化STEP:=20;
		END_IF
	20:
		IF 收集平台下压气缸原点 AND 收集平台夹持气缸原点
		   AND 收集平台升降气缸原点 AND 收集平台推出气缸原点
		   AND 泵初始化完成 THEN
			泵初始化完成:=FALSE;
			初始化STEP:=0;
			bActionDone:=TRUE;
		END_IF
END_CASE
END_ACTION

ACTION A42_伸缩缩回:
(* 搬运段2: 伸缩缩回 (上位机已先驱动机器人取瓶到暂存) *)
CASE 搬运step OF
	0:
		收集伸缩气缸自动:=FALSE;
		搬运step:=10;
	10:
		IF 收集平台推出气缸原点 THEN
			搬运step:=0;
			bActionDone:=TRUE;
		END_IF
END_CASE
END_ACTION

ACTION A41_复位伸出:
(* 搬运段1: 复位下压/升降 -> 伸缩伸出到取瓶位 *)
CASE 搬运step OF
	0:
		收集下压气缸自动:=FALSE;
		搬运step:=5;
	5:
		IF 收集平台下压气缸原点 THEN
			收集升降气缸自动:=FALSE;
			搬运step:=10;
		END_IF
	10:
		IF 收集平台升降气缸原点 THEN
			收集伸缩气缸自动:=TRUE;
			搬运step:=20;
		END_IF
	20:
		IF 收集平台推出气缸动点 THEN
			搬运step:=0;
			bActionDone:=TRUE;
		END_IF
END_CASE
END_ACTION

ACTION A43_松夹持:
(* 搬运段3: 松夹持 (上位机已先驱动机器人到收集器位) *)
CASE 搬运step OF
	0:
		收集夹持气缸自动:=FALSE;
		搬运step:=10;
	10:
		IF 收集平台夹持气缸原点 THEN
			搬运step:=0;
			bActionDone:=TRUE;
		END_IF
END_CASE
END_ACTION

END_PROGRAM

// Device/Application/30_Ethercat任务/PLC_Servo_伺服
PROGRAM PLC_Servo_伺服
VAR
	FB_SERVOAXIS_0: FB_SERVOAXIS;
	FB_SERVOAXIS_1: FB_SERVOAXIS;
	FB_SERVOAXIS_2: FB_SERVOAXIS;
	FB_SERVOAXIS_3: FB_SERVOAXIS;
	FB_SERVOAXIS_4: FB_SERVOAXIS;
	FB_SERVOAXIS_5: FB_SERVOAXIS;
	FB_SERVOAXIS_6: FB_SERVOAXIS;
	FB_SERVOAXIS_7: FB_SERVOAXIS;
	FB_SERVOAXIS_8: FB_SERVOAXIS;
	FB_SERVOAXIS_9: FB_SERVOAXIS;
	FB_SERVOAXIS_10: FB_SERVOAXIS;
	HOME_1STEP: INT;
	HOME_2STEP: INT;
	i: INT;
	FB_Teach_1: FB_Teach;
	FB_Teach_2: FB_Teach;
	FB_Teach_3: FB_Teach;
	FB_Teach_4: FB_Teach;
	FB_Teach_5: FB_Teach;
	FB_Teach_6: FB_Teach;
	n: INT;
	TON_SysReset: TON;
	bSysResetDone: BOOL;
	TON_CyInhibit: TON;
	bCyInhibitDone: BOOL;
	TON_AutoHome: TON;
	bAutoHomeDone: BOOL;
	TON_AutoHomeReset: TON;
	bAutoHomeReq: BOOL;
	bAutoHomeOnly45: BOOL;
	bAllHomed: BOOL;
	R_TRIG_HomeAll: R_TRIG;
	R_TRIG_Home45: R_TRIG;

	TON_BusStable: TON;
	TON_BusTimeout: TON;
	TON_ResetTimeout: TON;
	TON_EnableTimeout: TON;
	TON_RetreatTimeout: TON;
	TON_HomeTimeout: TON;
	TON_DeployPrepareTimeout: TON;
	R_TRIG_DeployStart: R_TRIG;
	bAllAxesComm: BOOL;
	bAllAxesEnabled: BOOL;
	bAnyAxisEnabled: BOOL;
	bAnyAxisBusy: BOOL;
	bAnyAxisErrorStop: BOOL;
	bAnyL2Busy: BOOL;
	bStartupResetIssued: BOOL;
	bAutoHome45Done: BOOL;

	bAnyAxisFault: BOOL;


	// CiA-402 0x60FD standard bits: 0 negative limit, 1 positive limit, 2 home switch.
	b5ZNegativeLimit: BOOL;
	b5ZPositiveLimit: BOOL;
	b5ZHomeSwitch: BOOL;
	b4XNegativeLimit: BOOL;
	b4XPositiveLimit: BOOL;
	b4XHomeSwitch: BOOL;
	b5ZRetreatUnsafe: BOOL;
	b4XRetreatUnsafe: BOOL;

	bAnyAuxOutputActive: BOOL;

END_VAR

// Compute alarm visibility before any axis/HMI-facing output.  Do not depend on
// initialization task ordering: the very first application scan must already be silent.
PLC_Startup_AlarmInhibit := ((NOT PLC_Ready) AND (PLC_Startup_State<>90))
	OR ((PLC_Deploy_State<>0) AND (PLC_Deploy_State<>30));

// Execute axis FBs first; command inputs are internally gated by communication/startup/maintenance state.
伺服调用();

PLC_Axis_CommOperational[1] := FB_SERVOAXIS_0.bCommOperational;
PLC_Axis_CommOperational[2] := FB_SERVOAXIS_1.bCommOperational;
PLC_Axis_CommOperational[3] := FB_SERVOAXIS_2.bCommOperational;
PLC_Axis_CommOperational[4] := FB_SERVOAXIS_3.bCommOperational;
PLC_Axis_CommOperational[5] := FB_SERVOAXIS_4.bCommOperational;
PLC_Axis_CommOperational[6] := FB_SERVOAXIS_5.bCommOperational;
PLC_Axis_CommOperational[7] := FB_SERVOAXIS_6.bCommOperational;
PLC_Axis_CommOperational[8] := FB_SERVOAXIS_7.bCommOperational;
PLC_Axis_CommOperational[9] := FB_SERVOAXIS_8.bCommOperational;
PLC_Axis_CommOperational[10] := FB_SERVOAXIS_9.bCommOperational;
PLC_Axis_CommOperational[11] := FB_SERVOAXIS_10.bCommOperational;
PLC_Axis_FaultSource[1] := FB_SERVOAXIS_0.iFaultSource; PLC_Axis_FaultCode[1] := FB_SERVOAXIS_0.iErrorCode;
PLC_Axis_FaultSource[2] := FB_SERVOAXIS_1.iFaultSource; PLC_Axis_FaultCode[2] := FB_SERVOAXIS_1.iErrorCode;
PLC_Axis_FaultSource[3] := FB_SERVOAXIS_2.iFaultSource; PLC_Axis_FaultCode[3] := FB_SERVOAXIS_2.iErrorCode;
PLC_Axis_FaultSource[4] := FB_SERVOAXIS_3.iFaultSource; PLC_Axis_FaultCode[4] := FB_SERVOAXIS_3.iErrorCode;
PLC_Axis_FaultSource[5] := FB_SERVOAXIS_4.iFaultSource; PLC_Axis_FaultCode[5] := FB_SERVOAXIS_4.iErrorCode;
PLC_Axis_FaultSource[6] := FB_SERVOAXIS_5.iFaultSource; PLC_Axis_FaultCode[6] := FB_SERVOAXIS_5.iErrorCode;
PLC_Axis_FaultSource[7] := FB_SERVOAXIS_6.iFaultSource; PLC_Axis_FaultCode[7] := FB_SERVOAXIS_6.iErrorCode;
PLC_Axis_FaultSource[8] := FB_SERVOAXIS_7.iFaultSource; PLC_Axis_FaultCode[8] := FB_SERVOAXIS_7.iErrorCode;
PLC_Axis_FaultSource[9] := FB_SERVOAXIS_8.iFaultSource; PLC_Axis_FaultCode[9] := FB_SERVOAXIS_8.iErrorCode;
PLC_Axis_FaultSource[10] := FB_SERVOAXIS_9.iFaultSource; PLC_Axis_FaultCode[10] := FB_SERVOAXIS_9.iErrorCode;
PLC_Axis_FaultSource[11] := FB_SERVOAXIS_10.iFaultSource; PLC_Axis_FaultCode[11] := FB_SERVOAXIS_10.iErrorCode;

bAllAxesComm := PLC_Axis_CommOperational[1] AND PLC_Axis_CommOperational[2]
	AND PLC_Axis_CommOperational[3] AND PLC_Axis_CommOperational[4]
	AND PLC_Axis_CommOperational[5] AND PLC_Axis_CommOperational[6]
	AND PLC_Axis_CommOperational[7] AND PLC_Axis_CommOperational[8]
	AND PLC_Axis_CommOperational[9] AND PLC_Axis_CommOperational[10]
	AND PLC_Axis_CommOperational[11];
bAllAxesEnabled := 玻璃上料轴1ZDATE.bEnabled AND 玻璃上料轴2ZDATE.bEnabled
	AND 打样瓶上料轴3YDATE.bEnabled AND 点样轴6XDATE.bEnabled AND 点样轴7YDATE.bEnabled
	AND 拍照轴8YDATE.bEnabled AND 刮板轴9XDATE.bEnabled AND 刮板轴10ZDATE.bEnabled
	AND 地轨轴11YDATE.bEnabled AND 上样轴4X轴DATE.bEnabled AND 上样轴5Z轴DATE.bEnabled;
bAnyAxisEnabled := 玻璃上料轴1ZDATE.bEnabled OR 玻璃上料轴2ZDATE.bEnabled
	OR 打样瓶上料轴3YDATE.bEnabled OR 点样轴6XDATE.bEnabled OR 点样轴7YDATE.bEnabled
	OR 拍照轴8YDATE.bEnabled OR 刮板轴9XDATE.bEnabled OR 刮板轴10ZDATE.bEnabled
	OR 地轨轴11YDATE.bEnabled OR 上样轴4X轴DATE.bEnabled OR 上样轴5Z轴DATE.bEnabled;
// 门禁"轴运动中"判据: 用 bMotionBusy (不含 MC_Power.Busy, 该位在使能期间恒为 TRUE) 而非聚合 bBusy;
// 速度阈值 1.0 mm/s: 实测空闲轴 fActVel 编码器量化噪声达 ±0.41 mm/s (0.0381 步进), 0.01 必然误报;
// 受控运动由 bMotionBusy 覆盖, 本阈值只兜未指令的外部/异常运动。
bAnyAxisBusy := FB_SERVOAXIS_0.bMotionBusy OR FB_SERVOAXIS_1.bMotionBusy
	OR FB_SERVOAXIS_2.bMotionBusy OR FB_SERVOAXIS_3.bMotionBusy
	OR FB_SERVOAXIS_4.bMotionBusy OR FB_SERVOAXIS_5.bMotionBusy
	OR FB_SERVOAXIS_6.bMotionBusy OR FB_SERVOAXIS_7.bMotionBusy
	OR FB_SERVOAXIS_8.bMotionBusy OR FB_SERVOAXIS_9.bMotionBusy
	OR FB_SERVOAXIS_10.bMotionBusy
	OR (ABS(玻璃上料轴1ZDATE.fActVel)>1.0) OR (ABS(玻璃上料轴2ZDATE.fActVel)>1.0)
	OR (ABS(打样瓶上料轴3YDATE.fActVel)>1.0) OR (ABS(点样轴6XDATE.fActVel)>1.0)
	OR (ABS(点样轴7YDATE.fActVel)>1.0) OR (ABS(拍照轴8YDATE.fActVel)>1.0)
	OR (ABS(刮板轴9XDATE.fActVel)>1.0) OR (ABS(刮板轴10ZDATE.fActVel)>1.0)
	OR (ABS(地轨轴11YDATE.fActVel)>1.0) OR (ABS(上样轴4X轴DATE.fActVel)>1.0)
	OR (ABS(上样轴5Z轴DATE.fActVel)>1.0) OR PLC_HandWheel_Active;
bAnyAxisErrorStop := (玻璃上料轴1Z.nAxisState=1) OR (玻璃上料轴2Z.nAxisState=1)
	OR (打样瓶上料轴3Y.nAxisState=1) OR (点样轴6X.nAxisState=1) OR (点样轴7Y.nAxisState=1)
	OR (拍照轴8Y.nAxisState=1) OR (刮板轴9X.nAxisState=1) OR (刮板轴10Z.nAxisState=1)
	OR (地轨轴11Y.nAxisState=1) OR (上样轴4X轴.nAxisState=1) OR (上样轴5Z轴.nAxisState=1);
bAnyAxisFault := FB_SERVOAXIS_0.bError OR FB_SERVOAXIS_1.bError OR FB_SERVOAXIS_2.bError
	OR FB_SERVOAXIS_3.bError OR FB_SERVOAXIS_4.bError OR FB_SERVOAXIS_5.bError
	OR FB_SERVOAXIS_6.bError OR FB_SERVOAXIS_7.bError OR FB_SERVOAXIS_8.bError
	OR FB_SERVOAXIS_9.bError OR FB_SERVOAXIS_10.bError;
b5ZNegativeLimit := (上样轴5Z轴.in.dwDigitalInputs AND DWORD#16#00000001) <> DWORD#0;
b5ZPositiveLimit := (上样轴5Z轴.in.dwDigitalInputs AND DWORD#16#00000002) <> DWORD#0;
b5ZHomeSwitch := (上样轴5Z轴.in.dwDigitalInputs AND DWORD#16#00000004) <> DWORD#0;
b4XNegativeLimit := (上样轴4X轴.in.dwDigitalInputs AND DWORD#16#00000001) <> DWORD#0;
b4XPositiveLimit := (上样轴4X轴.in.dwDigitalInputs AND DWORD#16#00000002) <> DWORD#0;
b4XHomeSwitch := (上样轴4X轴.in.dwDigitalInputs AND DWORD#16#00000004) <> DWORD#0;
b5ZRetreatUnsafe := b5ZPositiveLimit
	OR (上样轴5Z轴.bSWLimitEnable
		AND ((上样轴5Z轴DATE.fActPos + 10.0) > 上样轴5Z轴.fSWLimitPositive));
b4XRetreatUnsafe := b4XPositiveLimit
	OR (上样轴4X轴.bSWLimitEnable
		AND ((上样轴4X轴DATE.fActPos + 10.0) > 上样轴4X轴.fSWLimitPositive));
bAnyAuxOutputActive := 展缸1气缸1
	OR 展缸1气缸2
	OR 展缸1气缸3
	OR 展缸1气缸4
	OR 展缸2气缸1
	OR 展缸2气缸2
	OR 展缸2气缸3
	OR 展缸2气缸4
	OR 大真空泵
	OR 收集下压气缸
	OR 收集夹持气缸
	OR 收集升降气缸
	OR 收集伸缩气缸
	OR 刮板拍照遮光气缸
	OR 刮板拍照旋转气缸
	OR 刮板拍照下压气缸
	OR 展缸1进液电池阀1
	OR 展缸1进液电池阀2
	OR 展缸1进液电池阀3
	OR 展缸1进液电池阀4
	OR 展缸1排液电池阀1
	OR 展缸1排液电池阀2
	OR 展缸1排液电池阀3
	OR 展缸1排液电池阀4
	OR 展缸1吹气电池阀1
	OR 展缸1吹气电池阀2
	OR 展缸1吹气电池阀3
	OR 展缸1吹气电池阀4
	OR 展缸2进液电池阀1
	OR 展缸2进液电池阀2
	OR 展缸2进液电池阀3
	OR 展缸2进液电池阀4
	OR 展缸2排液电池阀1
	OR 展缸2排液电池阀2
	OR 展缸2排液电池阀3
	OR 展缸2排液电池阀4
	OR 展缸2吹气电池阀1
	OR 展缸2吹气电池阀2
	OR 展缸2吹气电池阀3
	OR 展缸2吹气电池阀4
	OR 收集平台进液2通电池阀
	OR 收集平台排液3通电池阀
	OR 收集平台正压排液阀
	OR 溶液收集瓶工位定位气缸
	OR 上样定位气缸
	OR 上样点样三通电池阀
	OR 刮板拍照真空阀
	OR 刮板拍照无刷电机
	OR 刮板拍照定位气缸
	OR 粉末收集器工位定位气缸
	OR 上样吹气二通阀
	OR 展缸1气缸1手动
	OR 展缸1气缸1自动
	OR 展缸1气缸2手动
	OR 展缸1气缸2自动
	OR 展缸1气缸3手动
	OR 展缸1气缸3自动
	OR 展缸1气缸4手动
	OR 展缸1气缸4自动
	OR 展缸2气缸1手动
	OR 展缸2气缸1自动
	OR 展缸2气缸2手动
	OR 展缸2气缸2自动
	OR 展缸2气缸3手动
	OR 展缸2气缸3自动
	OR 展缸2气缸4手动
	OR 展缸2气缸4自动
	OR 大真空泵手动
	OR 大真空泵自动
	OR 收集下压气缸手动
	OR 收集下压气缸自动
	OR 收集夹持气缸手动
	OR 收集夹持气缸自动
	OR 收集升降气缸手动
	OR 收集升降气缸自动
	OR 收集伸缩气缸手动
	OR 收集伸缩气缸自动
	OR 刮板拍照遮光气缸手动
	OR 刮板拍照遮光气缸自动
	OR 刮板拍照旋转气缸手动
	OR 刮板拍照旋转气缸自动
	OR 刮板拍照下压气缸手动
	OR 刮板拍照下压气缸自动
	OR 展缸1进液电池阀1手动
	OR 展缸1进液电池阀1自动
	OR 展缸1进液电池阀2手动
	OR 展缸1进液电池阀2自动
	OR 展缸1进液电池阀3手动
	OR 展缸1进液电池阀3自动
	OR 展缸1进液电池阀4手动
	OR 展缸1进液电池阀4自动
	OR 展缸1排液电池阀1手动
	OR 展缸1排液电池阀1自动
	OR 展缸1排液电池阀2手动
	OR 展缸1排液电池阀2自动
	OR 展缸1排液电池阀3手动
	OR 展缸1排液电池阀3自动
	OR 展缸1排液电池阀4手动
	OR 展缸1排液电池阀4自动
	OR 展缸1吹气电池阀1手动
	OR 展缸1吹气电池阀1自动
	OR 展缸1吹气电池阀2手动
	OR 展缸1吹气电池阀2自动
	OR 展缸1吹气电池阀3手动
	OR 展缸1吹气电池阀3自动
	OR 展缸1吹气电池阀4手动
	OR 展缸1吹气电池阀4自动
	OR 展缸2进液电池阀1手动
	OR 展缸2进液电池阀1自动
	OR 展缸2进液电池阀2手动
	OR 展缸2进液电池阀2自动
	OR 展缸2进液电池阀3手动
	OR 展缸2进液电池阀3自动
	OR 展缸2进液电池阀4手动
	OR 展缸2进液电池阀4自动
	OR 展缸2排液电池阀1手动
	OR 展缸2排液电池阀1自动
	OR 展缸2排液电池阀2手动
	OR 展缸2排液电池阀2自动
	OR 展缸2排液电池阀3手动
	OR 展缸2排液电池阀3自动
	OR 展缸2排液电池阀4手动
	OR 展缸2排液电池阀4自动
	OR 展缸2吹气电池阀1手动
	OR 展缸2吹气电池阀1自动
	OR 展缸2吹气电池阀2手动
	OR 展缸2吹气电池阀2自动
	OR 展缸2吹气电池阀3手动
	OR 展缸2吹气电池阀3自动
	OR 展缸2吹气电池阀4手动
	OR 展缸2吹气电池阀4自动
	OR 收集进液手动
	OR 收集进液自动
	OR 收集排液手动
	OR 收集排液自动
	OR 收集正压排液手动
	OR 收集正压排液自动
	OR 溶液收集瓶定位手动
	OR 溶液收集瓶定位自动
	OR 上样定位手动
	OR 上样定位自动
	OR 上样点样三通电池阀手动
	OR 上样点样三通电池阀自动
	OR 刮板拍照真空手动
	OR 刮板拍照真空自动
	OR 刮板拍照无刷电机手动
	OR 刮板拍照无刷电机自动
	OR 刮板拍照定位气缸手动
	OR 刮板拍照定位气缸自动
	OR 粉末收集器定位手动
	OR 粉末收集器定位自动
	OR 上样吹气手动
	OR 上样吹气自动
	OR 大真空泵站位[0]
	OR 大真空泵站位[1]
	OR 大真空泵站位[2]
	OR 大真空泵站位[3]
	OR 大真空泵站位[4]
	OR 大真空泵站位[5]
	OR 大真空泵站位[6]
	OR 大真空泵站位[7]
	OR 大真空泵站位[8]
	OR 大真空泵站位[9]
	OR 大真空泵站位[10]
	OR 大真空泵站位[11]
	OR Tank_Drain_Enable[1]
	OR ((Tank_State[1]=50) OR (Tank_State[1]=55) OR (Tank_State[1]=56))
	OR Tank_Drain_Enable[2]
	OR ((Tank_State[2]=50) OR (Tank_State[2]=55) OR (Tank_State[2]=56))
	OR Tank_Drain_Enable[3]
	OR ((Tank_State[3]=50) OR (Tank_State[3]=55) OR (Tank_State[3]=56))
	OR Tank_Drain_Enable[4]
	OR ((Tank_State[4]=50) OR (Tank_State[4]=55) OR (Tank_State[4]=56))
	OR Tank_Drain_Enable[5]
	OR ((Tank_State[5]=50) OR (Tank_State[5]=55) OR (Tank_State[5]=56))
	OR Tank_Drain_Enable[6]
	OR ((Tank_State[6]=50) OR (Tank_State[6]=55) OR (Tank_State[6]=56))
	OR Tank_Drain_Enable[7]
	OR ((Tank_State[7]=50) OR (Tank_State[7]=55) OR (Tank_State[7]=56))
	OR Tank_Drain_Enable[8]
	OR ((Tank_State[8]=50) OR (Tank_State[8]=55) OR (Tank_State[8]=56))
	OR 泵站位符
	OR (%MW1300<>0);
bAnyL2Busy := (Collect_L2_State=10) OR (Sampling_L2_State=10) OR (Develop_L2_State=10)
	OR (PhotoScrape_L2_State=10) OR (FeedLift_L2_State=10) OR (Pump_L2_State=10)
	OR (Rail_L2_State=10) OR (StagingA_L2_State=10);

// Download prepare handshake. A busy machine is rejected; running actions are never interrupted.
R_TRIG_DeployStart(CLK := PLC_Deploy_Start);
TON_DeployPrepareTimeout(IN := PLC_Deploy_State=10, PT := T#10S);
IF PLC_Deploy_Reset AND NOT PLC_Deploy_Start
	AND ((PLC_Deploy_State<>25) OR (PLC_Deploy_CommitSeq=0)) THEN
	PLC_Deploy_State := 0;
	PLC_Deploy_ErrorCode := 0;
ELSIF R_TRIG_DeployStart.Q AND PLC_Deploy_State=0 THEN
	PLC_Deploy_AcceptedSeq := PLC_Deploy_RequestSeq;
	IF bAnyL2Busy THEN
		PLC_Deploy_State := 30; PLC_Deploy_ErrorCode := 1;
	ELSIF bAnyAxisBusy THEN
		PLC_Deploy_State := 30; PLC_Deploy_ErrorCode := 2;
	ELSIF bAnyAuxOutputActive THEN
		PLC_Deploy_State := 30; PLC_Deploy_ErrorCode := 3;
	ELSIF NOT PLC_Ready OR NOT bAllAxesComm THEN
		PLC_Deploy_State := 40; PLC_Deploy_ErrorCode := 5;
	ELSE
		玻璃上料轴1ZDATE.xHome := FALSE; 玻璃上料轴1ZDATE.xJogPos := FALSE; 玻璃上料轴1ZDATE.xJogNeg := FALSE;
		玻璃上料轴1ZDATE.xMoveAbs := FALSE; 玻璃上料轴1ZDATE.xMoveRel := FALSE; 玻璃上料轴1ZDATE.xStop := FALSE; 玻璃上料轴1ZDATE.XReset := FALSE;
		玻璃上料轴2ZDATE.xHome := FALSE; 玻璃上料轴2ZDATE.xJogPos := FALSE; 玻璃上料轴2ZDATE.xJogNeg := FALSE;
		玻璃上料轴2ZDATE.xMoveAbs := FALSE; 玻璃上料轴2ZDATE.xMoveRel := FALSE; 玻璃上料轴2ZDATE.xStop := FALSE; 玻璃上料轴2ZDATE.XReset := FALSE;
		打样瓶上料轴3YDATE.xHome := FALSE; 打样瓶上料轴3YDATE.xJogPos := FALSE; 打样瓶上料轴3YDATE.xJogNeg := FALSE;
		打样瓶上料轴3YDATE.xMoveAbs := FALSE; 打样瓶上料轴3YDATE.xMoveRel := FALSE; 打样瓶上料轴3YDATE.xStop := FALSE; 打样瓶上料轴3YDATE.XReset := FALSE;
		点样轴6XDATE.xHome := FALSE; 点样轴6XDATE.xJogPos := FALSE; 点样轴6XDATE.xJogNeg := FALSE;
		点样轴6XDATE.xMoveAbs := FALSE; 点样轴6XDATE.xMoveRel := FALSE; 点样轴6XDATE.xStop := FALSE; 点样轴6XDATE.XReset := FALSE;
		点样轴7YDATE.xHome := FALSE; 点样轴7YDATE.xJogPos := FALSE; 点样轴7YDATE.xJogNeg := FALSE;
		点样轴7YDATE.xMoveAbs := FALSE; 点样轴7YDATE.xMoveRel := FALSE; 点样轴7YDATE.xStop := FALSE; 点样轴7YDATE.XReset := FALSE;
		拍照轴8YDATE.xHome := FALSE; 拍照轴8YDATE.xJogPos := FALSE; 拍照轴8YDATE.xJogNeg := FALSE;
		拍照轴8YDATE.xMoveAbs := FALSE; 拍照轴8YDATE.xMoveRel := FALSE; 拍照轴8YDATE.xStop := FALSE; 拍照轴8YDATE.XReset := FALSE;
		刮板轴9XDATE.xHome := FALSE; 刮板轴9XDATE.xJogPos := FALSE; 刮板轴9XDATE.xJogNeg := FALSE;
		刮板轴9XDATE.xMoveAbs := FALSE; 刮板轴9XDATE.xMoveRel := FALSE; 刮板轴9XDATE.xStop := FALSE; 刮板轴9XDATE.XReset := FALSE;
		刮板轴10ZDATE.xHome := FALSE; 刮板轴10ZDATE.xJogPos := FALSE; 刮板轴10ZDATE.xJogNeg := FALSE;
		刮板轴10ZDATE.xMoveAbs := FALSE; 刮板轴10ZDATE.xMoveRel := FALSE; 刮板轴10ZDATE.xStop := FALSE; 刮板轴10ZDATE.XReset := FALSE;
		地轨轴11YDATE.xHome := FALSE; 地轨轴11YDATE.xJogPos := FALSE; 地轨轴11YDATE.xJogNeg := FALSE;
		地轨轴11YDATE.xMoveAbs := FALSE; 地轨轴11YDATE.xMoveRel := FALSE; 地轨轴11YDATE.xStop := FALSE; 地轨轴11YDATE.XReset := FALSE;
		上样轴4X轴DATE.xHome := FALSE; 上样轴4X轴DATE.xJogPos := FALSE; 上样轴4X轴DATE.xJogNeg := FALSE;
		上样轴4X轴DATE.xMoveAbs := FALSE; 上样轴4X轴DATE.xMoveRel := FALSE; 上样轴4X轴DATE.xStop := FALSE; 上样轴4X轴DATE.XReset := FALSE;
		上样轴5Z轴DATE.xHome := FALSE; 上样轴5Z轴DATE.xJogPos := FALSE; 上样轴5Z轴DATE.xJogNeg := FALSE;
		上样轴5Z轴DATE.xMoveAbs := FALSE; 上样轴5Z轴DATE.xMoveRel := FALSE; 上样轴5Z轴DATE.xStop := FALSE; 上样轴5Z轴DATE.XReset := FALSE;
		PLC_Deploy_ErrorCode := 0;
		PLC_Deploy_State := 10;
	END_IF
ELSIF PLC_Deploy_State=10 THEN
	IF (ethercat1.m_master.m_uiactualnoslaves<>13) OR (ethercat1.m_master._masterState<>8) OR NOT bAllAxesComm THEN
		PLC_Deploy_State := 40; PLC_Deploy_ErrorCode := 5;
	ELSIF bAnyAuxOutputActive THEN
		PLC_Deploy_State := 40; PLC_Deploy_ErrorCode := 42;
	ELSIF NOT bAnyAxisEnabled AND NOT bAnyAxisBusy THEN
		PLC_Deploy_State := 20;
	ELSIF TON_DeployPrepareTimeout.Q THEN
		PLC_Deploy_State := 40; PLC_Deploy_ErrorCode := 40;
	END_IF
ELSIF PLC_Deploy_State=20 THEN
	// READY_TO_DOWNLOAD is a maintained invariant, not a one-scan acknowledgement.
	IF (ethercat1.m_master.m_uiactualnoslaves<>13) OR (ethercat1.m_master._masterState<>8) OR NOT bAllAxesComm THEN
		PLC_Deploy_State := 40; PLC_Deploy_ErrorCode := 5;
	ELSIF bAnyAxisEnabled OR bAnyAxisBusy OR PLC_HandWheel_Active OR bAnyAuxOutputActive THEN
		PLC_Deploy_State := 40; PLC_Deploy_ErrorCode := 41;
	ELSIF PLC_Deploy_Start AND (PLC_Deploy_CommitSeq=PLC_Deploy_AcceptedSeq)
		AND (PLC_Deploy_CommitSeq<>0) THEN
		PLC_Deploy_State := 25;
	END_IF
ELSIF PLC_Deploy_State=25 THEN
	// Host committed: normal HMI Start/Reset cancellation is ignored until a confirmed
	// pre-download abort explicitly clears CommitSeq. Full download reinitialises the application.
	IF (ethercat1.m_master.m_uiactualnoslaves<>13) OR (ethercat1.m_master._masterState<>8) OR NOT bAllAxesComm THEN
		PLC_Deploy_ErrorCode := 5;
	ELSIF bAnyAxisEnabled OR bAnyAxisBusy OR PLC_HandWheel_Active OR bAnyAuxOutputActive THEN
		PLC_Deploy_ErrorCode := 41;
	END_IF
END_IF

// Startup timers. Safety-chain wait itself is intentionally untimed; no motion begins until it is healthy.
TON_BusStable(IN := PLC_Startup_State=10 AND ethercat1.m_master.m_uiactualnoslaves=13
	AND (ethercat1.m_master._masterState=8) AND bAllAxesComm, PT := T#2S);
TON_BusTimeout(IN := PLC_Startup_State=10, PT := T#30S);
TON_ResetTimeout(IN := PLC_Startup_State=20 AND 急停 AND bStartupResetIssued
	AND (bAnyAxisErrorStop OR bAnyAxisFault), PT := T#5S);
TON_EnableTimeout(IN := PLC_Startup_State=30 AND 急停 AND NOT bAllAxesEnabled, PT := T#10S);
TON_RetreatTimeout(IN := (PLC_Startup_State=40) OR (PLC_Startup_State=50), PT := T#15S);
TON_HomeTimeout(IN := (PLC_Startup_State=41) OR (PLC_Startup_State=51), PT := T#60S);

bSysReset := FALSE;
IF 复位 AND PLC_Startup_State=90 THEN
	PLC_Startup_State := 0;
END_IF

// Once EtherCAT startup has succeeded, a later bus/axis-communication loss is always the root cause.
// It outranks reset, enable and homing timeouts and is never treated as eleven independent servo faults.
IF (PLC_Startup_State>=20) AND (PLC_Startup_State<=60)
	AND ((ethercat1.m_master.m_uiactualnoslaves<>13) OR (ethercat1.m_master._masterState<>8) OR NOT bAllAxesComm) THEN
	PLC_Ready := FALSE;
	PLC_Startup_ErrorCode := 100;
	PLC_Startup_State := 90;
END_IF

CASE PLC_Startup_State OF
	0:
		PLC_Ready := FALSE;
		PLC_Startup_ErrorCode := 0;
		bStartupResetIssued := FALSE;
		bAutoHomeReq := FALSE;
		HOME_2STEP := 0;
		PLC_HandWheel_Active := FALSE;
		玻璃上料轴1ZDATE.xHome := FALSE; 玻璃上料轴1ZDATE.xJogPos := FALSE; 玻璃上料轴1ZDATE.xJogNeg := FALSE;
		玻璃上料轴1ZDATE.xMoveAbs := FALSE; 玻璃上料轴1ZDATE.xMoveRel := FALSE; 玻璃上料轴1ZDATE.xStop := FALSE; 玻璃上料轴1ZDATE.XReset := FALSE;
		玻璃上料轴2ZDATE.xHome := FALSE; 玻璃上料轴2ZDATE.xJogPos := FALSE; 玻璃上料轴2ZDATE.xJogNeg := FALSE;
		玻璃上料轴2ZDATE.xMoveAbs := FALSE; 玻璃上料轴2ZDATE.xMoveRel := FALSE; 玻璃上料轴2ZDATE.xStop := FALSE; 玻璃上料轴2ZDATE.XReset := FALSE;
		打样瓶上料轴3YDATE.xHome := FALSE; 打样瓶上料轴3YDATE.xJogPos := FALSE; 打样瓶上料轴3YDATE.xJogNeg := FALSE;
		打样瓶上料轴3YDATE.xMoveAbs := FALSE; 打样瓶上料轴3YDATE.xMoveRel := FALSE; 打样瓶上料轴3YDATE.xStop := FALSE; 打样瓶上料轴3YDATE.XReset := FALSE;
		点样轴6XDATE.xHome := FALSE; 点样轴6XDATE.xJogPos := FALSE; 点样轴6XDATE.xJogNeg := FALSE;
		点样轴6XDATE.xMoveAbs := FALSE; 点样轴6XDATE.xMoveRel := FALSE; 点样轴6XDATE.xStop := FALSE; 点样轴6XDATE.XReset := FALSE;
		点样轴7YDATE.xHome := FALSE; 点样轴7YDATE.xJogPos := FALSE; 点样轴7YDATE.xJogNeg := FALSE;
		点样轴7YDATE.xMoveAbs := FALSE; 点样轴7YDATE.xMoveRel := FALSE; 点样轴7YDATE.xStop := FALSE; 点样轴7YDATE.XReset := FALSE;
		拍照轴8YDATE.xHome := FALSE; 拍照轴8YDATE.xJogPos := FALSE; 拍照轴8YDATE.xJogNeg := FALSE;
		拍照轴8YDATE.xMoveAbs := FALSE; 拍照轴8YDATE.xMoveRel := FALSE; 拍照轴8YDATE.xStop := FALSE; 拍照轴8YDATE.XReset := FALSE;
		刮板轴9XDATE.xHome := FALSE; 刮板轴9XDATE.xJogPos := FALSE; 刮板轴9XDATE.xJogNeg := FALSE;
		刮板轴9XDATE.xMoveAbs := FALSE; 刮板轴9XDATE.xMoveRel := FALSE; 刮板轴9XDATE.xStop := FALSE; 刮板轴9XDATE.XReset := FALSE;
		刮板轴10ZDATE.xHome := FALSE; 刮板轴10ZDATE.xJogPos := FALSE; 刮板轴10ZDATE.xJogNeg := FALSE;
		刮板轴10ZDATE.xMoveAbs := FALSE; 刮板轴10ZDATE.xMoveRel := FALSE; 刮板轴10ZDATE.xStop := FALSE; 刮板轴10ZDATE.XReset := FALSE;
		地轨轴11YDATE.xHome := FALSE; 地轨轴11YDATE.xJogPos := FALSE; 地轨轴11YDATE.xJogNeg := FALSE;
		地轨轴11YDATE.xMoveAbs := FALSE; 地轨轴11YDATE.xMoveRel := FALSE; 地轨轴11YDATE.xStop := FALSE; 地轨轴11YDATE.XReset := FALSE;
		上样轴4X轴DATE.xHome := FALSE; 上样轴4X轴DATE.xJogPos := FALSE; 上样轴4X轴DATE.xJogNeg := FALSE;
		上样轴4X轴DATE.xMoveAbs := FALSE; 上样轴4X轴DATE.xMoveRel := FALSE; 上样轴4X轴DATE.xStop := FALSE; 上样轴4X轴DATE.XReset := FALSE;
		上样轴5Z轴DATE.xHome := FALSE; 上样轴5Z轴DATE.xJogPos := FALSE; 上样轴5Z轴DATE.xJogNeg := FALSE;
		上样轴5Z轴DATE.xMoveAbs := FALSE; 上样轴5Z轴DATE.xMoveRel := FALSE; 上样轴5Z轴DATE.xStop := FALSE; 上样轴5Z轴DATE.XReset := FALSE;
		上样轴5Z轴DATE.bHomed := FALSE;
		上样轴4X轴DATE.bHomed := FALSE;
		PLC_Startup_State := 10;
	10:
		PLC_Ready := FALSE;
		IF TON_BusStable.Q THEN
			bStartupResetIssued := FALSE;
			PLC_Startup_State := 20;
		ELSIF TON_BusTimeout.Q THEN
			IF (ethercat1.m_master.m_uiactualnoslaves<>13) OR (ethercat1.m_master._masterState<>8) THEN
				PLC_Startup_ErrorCode := 100;
			ELSE
				PLC_Startup_ErrorCode := 200;
			END_IF
			PLC_Startup_State := 90;
		END_IF
	20:
		IF 急停 THEN
			IF NOT bStartupResetIssued THEN
				bSysReset := TRUE;
				bStartupResetIssued := TRUE;
			ELSIF NOT bAnyAxisErrorStop AND NOT bAnyAxisFault THEN
				PLC_Startup_State := 30;
			ELSIF TON_ResetTimeout.Q THEN
				PLC_Startup_ErrorCode := 300;
				PLC_Startup_State := 90;
			END_IF
		END_IF
	30:
		IF 急停 THEN
			IF bAnyAxisFault THEN
				PLC_Startup_ErrorCode := 301;
				PLC_Startup_State := 90;
			ELSIF bAllAxesEnabled THEN
				bAutoHomeReq := TRUE;
				PLC_Startup_State := 40;
			ELSIF TON_EnableTimeout.Q THEN
				PLC_Startup_ErrorCode := 400;
				PLC_Startup_State := 90;
			END_IF
		END_IF
	40:
		IF NOT 急停 THEN
			PLC_Startup_ErrorCode := 900; PLC_Startup_State := 90;
		ELSIF b5ZRetreatUnsafe THEN
			PLC_Startup_ErrorCode := 515; PLC_Startup_State := 90;
		ELSIF FB_SERVOAXIS_10.bError THEN
			PLC_Startup_ErrorCode := 705; PLC_Startup_State := 90;
		ELSIF bAnyAxisFault THEN
			PLC_Startup_ErrorCode := 301; PLC_Startup_State := 90;
		ELSIF HOME_2STEP=4 THEN
			PLC_Startup_State := 41;
		ELSIF TON_RetreatTimeout.Q THEN
			PLC_Startup_ErrorCode := 505; PLC_Startup_State := 90;
		END_IF
	41:
		IF NOT 急停 THEN
			PLC_Startup_ErrorCode := 900; PLC_Startup_State := 90;
		ELSIF (HOME_2STEP=4) AND 上样轴5Z轴DATE.bHomed AND b4XRetreatUnsafe THEN
			PLC_Startup_ErrorCode := 514; PLC_Startup_State := 90;
		ELSIF FB_SERVOAXIS_10.bError THEN
			PLC_Startup_ErrorCode := 705; PLC_Startup_State := 90;
		ELSIF bAnyAxisFault THEN
			PLC_Startup_ErrorCode := 301; PLC_Startup_State := 90;
		ELSIF HOME_2STEP=5 THEN
			PLC_Startup_State := 50;
		ELSIF TON_HomeTimeout.Q THEN
			PLC_Startup_ErrorCode := 605; PLC_Startup_State := 90;
		END_IF
	50:
		IF NOT 急停 THEN
			PLC_Startup_ErrorCode := 900; PLC_Startup_State := 90;
		ELSIF b4XRetreatUnsafe THEN
			PLC_Startup_ErrorCode := 514; PLC_Startup_State := 90;
		ELSIF FB_SERVOAXIS_9.bError THEN
			PLC_Startup_ErrorCode := 704; PLC_Startup_State := 90;
		ELSIF bAnyAxisFault THEN
			PLC_Startup_ErrorCode := 301; PLC_Startup_State := 90;
		ELSIF HOME_2STEP=6 THEN
			PLC_Startup_State := 51;
		ELSIF TON_RetreatTimeout.Q THEN
			PLC_Startup_ErrorCode := 504; PLC_Startup_State := 90;
		END_IF
	51:
		IF NOT 急停 THEN
			PLC_Startup_ErrorCode := 900; PLC_Startup_State := 90;
		ELSIF FB_SERVOAXIS_9.bError THEN
			PLC_Startup_ErrorCode := 704; PLC_Startup_State := 90;
		ELSIF bAnyAxisFault THEN
			PLC_Startup_ErrorCode := 301; PLC_Startup_State := 90;
		ELSIF (HOME_2STEP=0) AND 上样轴5Z轴DATE.bHomed AND 上样轴4X轴DATE.bHomed THEN
			PLC_Startup_State := 60;
		ELSIF TON_HomeTimeout.Q THEN
			PLC_Startup_ErrorCode := 604; PLC_Startup_State := 90;
		END_IF
	60:
		IF NOT 急停 THEN
			PLC_Ready := FALSE;
			PLC_Startup_ErrorCode := 900;
			PLC_Startup_State := 90;
		ELSIF bAnyAxisFault THEN
			PLC_Ready := FALSE;
			PLC_Startup_ErrorCode := 301;
			PLC_Startup_State := 90;
		ELSE
			PLC_Ready := bAllAxesEnabled
				AND ((PLC_Deploy_State=0) OR (PLC_Deploy_State=30));
		END_IF
	90:
		PLC_Ready := FALSE;
		bAutoHomeReq := FALSE;
		HOME_2STEP := 0;
		玻璃上料轴1ZDATE.xStop := TRUE;
		玻璃上料轴2ZDATE.xStop := TRUE;
		打样瓶上料轴3YDATE.xStop := TRUE;
		点样轴6XDATE.xStop := TRUE;
		点样轴7YDATE.xStop := TRUE;
		拍照轴8YDATE.xStop := TRUE;
		刮板轴9XDATE.xStop := TRUE;
		刮板轴10ZDATE.xStop := TRUE;
		地轨轴11YDATE.xStop := TRUE;
		上样轴4X轴DATE.xStop := TRUE;
		上样轴5Z轴DATE.xStop := TRUE;
		上样轴5Z轴DATE.xHome := FALSE;
		上样轴5Z轴DATE.xMoveRel := FALSE;
		上样轴4X轴DATE.xHome := FALSE;
		上样轴4X轴DATE.xMoveRel := FALSE;
END_CASE

bSysResetDone := PLC_Startup_State>=30 AND PLC_Startup_State<>90;
bAutoHome45Done := 上样轴5Z轴DATE.bHomed AND 上样轴4X轴DATE.bHomed;
IF bAutoHomeReq AND bAutoHome45Done THEN
	TON_AutoHomeReset(IN := TRUE, PT := T#1500MS);
	bAutoHomeResetPulse := TRUE;
	IF TON_AutoHomeReset.Q THEN
		bAutoHomeReq := FALSE;
		bAutoHomeResetPulse := FALSE;
	END_IF
ELSE
	TON_AutoHomeReset(IN := FALSE, PT := T#1500MS);
	bAutoHomeResetPulse := FALSE;
END_IF

// Keep the existing cylinder startup suppression window.
TON_CyInhibit(IN := ethercat1.m_master.m_uiactualnoslaves=13 AND NOT bCyInhibitDone, PT := T#15S);
bCyInhibit := (ethercat1.m_master.m_uiactualnoslaves=13) AND NOT bCyInhibitDone;
IF TON_CyInhibit.Q THEN bCyInhibitDone := TRUE; END_IF

// Refresh alarm visibility before every alarm outlet.  The same expression is also evaluated at
// the very top of this POU before the axis calls, so a fresh download cannot leak a first-scan pulse.
PLC_Startup_AlarmInhibit := ((NOT PLC_Ready) AND (PLC_Startup_State<>90))
	OR ((PLC_Deploy_State<>0) AND (PLC_Deploy_State<>30));

// Successful initialization is silent. Only a terminal startup failure or a post-ready loss is alarmed.
IF PLC_Startup_AlarmInhibit THEN
	ECAT掉站报警 := FALSE;
ELSIF (PLC_Startup_State=90) AND (PLC_Startup_ErrorCode>=100) AND (PLC_Startup_ErrorCode<=200) THEN
	ECAT掉站报警 := TRUE;
ELSE
	ECAT掉站报警 := (ethercat1.m_master.m_uiactualnoslaves<>13) OR (ethercat1.m_master._masterState<>8);
END_IF

// Retained/HMI motion requests are continuously drained while startup or maintenance owns motion.
// The automatic homing POU below reasserts only the currently authorised 5Z/4X command.
IF (NOT PLC_Ready) OR ((PLC_Deploy_State<>0) AND (PLC_Deploy_State<>30)) THEN
	玻璃上料轴1ZDATE.xHome := FALSE; 玻璃上料轴1ZDATE.xJogPos := FALSE; 玻璃上料轴1ZDATE.xJogNeg := FALSE;
	玻璃上料轴1ZDATE.xMoveAbs := FALSE; 玻璃上料轴1ZDATE.xMoveRel := FALSE; 玻璃上料轴1ZDATE.XReset := FALSE;
	玻璃上料轴2ZDATE.xHome := FALSE; 玻璃上料轴2ZDATE.xJogPos := FALSE; 玻璃上料轴2ZDATE.xJogNeg := FALSE;
	玻璃上料轴2ZDATE.xMoveAbs := FALSE; 玻璃上料轴2ZDATE.xMoveRel := FALSE; 玻璃上料轴2ZDATE.XReset := FALSE;
	打样瓶上料轴3YDATE.xHome := FALSE; 打样瓶上料轴3YDATE.xJogPos := FALSE; 打样瓶上料轴3YDATE.xJogNeg := FALSE;
	打样瓶上料轴3YDATE.xMoveAbs := FALSE; 打样瓶上料轴3YDATE.xMoveRel := FALSE; 打样瓶上料轴3YDATE.XReset := FALSE;
	点样轴6XDATE.xHome := FALSE; 点样轴6XDATE.xJogPos := FALSE; 点样轴6XDATE.xJogNeg := FALSE;
	点样轴6XDATE.xMoveAbs := FALSE; 点样轴6XDATE.xMoveRel := FALSE; 点样轴6XDATE.XReset := FALSE;
	点样轴7YDATE.xHome := FALSE; 点样轴7YDATE.xJogPos := FALSE; 点样轴7YDATE.xJogNeg := FALSE;
	点样轴7YDATE.xMoveAbs := FALSE; 点样轴7YDATE.xMoveRel := FALSE; 点样轴7YDATE.XReset := FALSE;
	拍照轴8YDATE.xHome := FALSE; 拍照轴8YDATE.xJogPos := FALSE; 拍照轴8YDATE.xJogNeg := FALSE;
	拍照轴8YDATE.xMoveAbs := FALSE; 拍照轴8YDATE.xMoveRel := FALSE; 拍照轴8YDATE.XReset := FALSE;
	刮板轴9XDATE.xHome := FALSE; 刮板轴9XDATE.xJogPos := FALSE; 刮板轴9XDATE.xJogNeg := FALSE;
	刮板轴9XDATE.xMoveAbs := FALSE; 刮板轴9XDATE.xMoveRel := FALSE; 刮板轴9XDATE.XReset := FALSE;
	刮板轴10ZDATE.xHome := FALSE; 刮板轴10ZDATE.xJogPos := FALSE; 刮板轴10ZDATE.xJogNeg := FALSE;
	刮板轴10ZDATE.xMoveAbs := FALSE; 刮板轴10ZDATE.xMoveRel := FALSE; 刮板轴10ZDATE.XReset := FALSE;
	地轨轴11YDATE.xHome := FALSE; 地轨轴11YDATE.xJogPos := FALSE; 地轨轴11YDATE.xJogNeg := FALSE;
	地轨轴11YDATE.xMoveAbs := FALSE; 地轨轴11YDATE.xMoveRel := FALSE; 地轨轴11YDATE.XReset := FALSE;
	上样轴4X轴DATE.xHome := FALSE; 上样轴4X轴DATE.xJogPos := FALSE; 上样轴4X轴DATE.xJogNeg := FALSE;
	上样轴4X轴DATE.xMoveAbs := FALSE; 上样轴4X轴DATE.xMoveRel := FALSE; 上样轴4X轴DATE.XReset := FALSE;
	上样轴5Z轴DATE.xHome := FALSE; 上样轴5Z轴DATE.xJogPos := FALSE; 上样轴5Z轴DATE.xJogNeg := FALSE;
	上样轴5Z轴DATE.xMoveAbs := FALSE; 上样轴5Z轴DATE.xMoveRel := FALSE; 上样轴5Z轴DATE.XReset := FALSE;
	Z1JOG_pos := FALSE;
	Z1JOG_neg := FALSE;
	Z2JOG_POS := FALSE;
	Z2JOG_NEG := FALSE;
	Sampling_Servo_FreeMove := FALSE;
END_IF

// The six teaching arrays are RETAIN PERSISTENT command sources. Clearing only the
// derived axis command is insufficient because 位置示教 can recreate it later. Drain
// both execute/write sources every scan while startup or maintenance owns motion.
IF (NOT PLC_Ready) OR ((PLC_Deploy_State<>0) AND (PLC_Deploy_State<>30)) THEN
	FOR n:=1 TO 10 DO
		HMI_打样瓶上料轴3Y.execute[n] := FALSE;
		HMI_打样瓶上料轴3Y.write[n] := FALSE;
		HMI_点样轴6X.execute[n] := FALSE;
		HMI_点样轴6X.write[n] := FALSE;
		HMI_点样轴7Y.execute[n] := FALSE;
		HMI_点样轴7Y.write[n] := FALSE;
		HMI_地轨轴11Y.execute[n] := FALSE;
		HMI_地轨轴11Y.write[n] := FALSE;
		HMI_上样轴4X轴.execute[n] := FALSE;
		HMI_上样轴4X轴.write[n] := FALSE;
		HMI_上样轴5Z轴.execute[n] := FALSE;
		HMI_上样轴5Z轴.write[n] := FALSE;
	END_FOR
	一键回原点 := FALSE;
END_IF

IF ((MODE_State<>1) AND PLC_Ready)
	OR ((PLC_Startup_State>=40) AND (PLC_Startup_State<=51)) THEN
	伺服一键回原点();
END_IF
IF PLC_Ready
	AND ((PLC_Deploy_State=0) OR (PLC_Deploy_State=30))
	AND (MODE_State<>1) AND NOT 点样测试 THEN
	位置示教();
END_IF

IF MODE_State=1 THEN		
	FOR n:=1 TO 10 BY 1 DO
		HMI_打样瓶上料轴3Y.execute[n]:=FALSE;
		HMI_打样瓶上料轴3Y.write[n]:=FALSE;
		HMI_点样轴6X.execute[n]:=FALSE;
		HMI_点样轴6X.write[n]:=FALSE;
		HMI_点样轴7Y.execute[n]:=FALSE;
		HMI_点样轴7Y.write[n]:=FALSE;
		HMI_地轨轴11Y.execute[n]:=FALSE;
		HMI_地轨轴11Y.write[n]:=FALSE;
		HMI_上样轴4X轴.execute[n]:=FALSE;
		HMI_上样轴4X轴.write[n]:=FALSE;
		HMI_上样轴5Z轴.execute[n]:=FALSE;
		HMI_上样轴5Z轴.write[n]:=FALSE;	
	END_FOR
		HMI_HandWheel_3Y:=FALSE;
		HMI_HandWheel_4X:=FALSE;
		HMI_HandWheel_5Z:=FALSE;
		HMI_HandWheel_6X:=FALSE;
		HMI_HandWheel_7Y:=FALSE;
		HMI_HandWheel_8Y:=FALSE;
		HMI_HandWheel_9X:=FALSE;
		HMI_HandWheel_10Z:=FALSE;
		HMI_HandWheel_11Y:=FALSE;

	
END_IF

ACTION 伺服一键回原点:
// Manual request homes all axes; startup request homes only incremental 5Z then 4X.
// PC 单点控制 (PLC_PCManual.PC_Manual_Active) 与柜面手动档等价放行: 该模式下
// MODE_State<>运行 且 8 工位 L2 全空闲已由 PLC_PCManual 保证, 安全前提与手动档一致。
R_TRIG_HomeAll(CLK := 一键回原点 AND PLC_Ready AND ((PLC_Deploy_State=0) OR (PLC_Deploy_State=30)) AND MODE_State<>1 AND (NOT ManualAuto OR PLC_PCManual.PC_Manual_Active));
R_TRIG_Home45(CLK := bAutoHomeReq);

IF R_TRIG_HomeAll.Q THEN
	玻璃上料轴1ZDATE.bHomed := FALSE; 玻璃上料轴1ZDATE.xHome := TRUE;
	玻璃上料轴2ZDATE.bHomed := FALSE; 玻璃上料轴2ZDATE.xHome := TRUE;
	刮板轴10ZDATE.bHomed := FALSE; 刮板轴10ZDATE.xHome := TRUE;
	点样轴6XDATE.bHomed := FALSE; 点样轴6XDATE.xHome := TRUE;
	点样轴7YDATE.bHomed := FALSE; 点样轴7YDATE.xHome := TRUE;
	地轨轴11YDATE.bHomed := FALSE; 地轨轴11YDATE.xHome := TRUE;
	HOME_1STEP := 1;
	HOME_2STEP := 1;
	bAutoHomeOnly45 := FALSE;
END_IF

IF R_TRIG_Home45.Q THEN
	上样轴5Z轴DATE.bHomed := FALSE;
	上样轴4X轴DATE.bHomed := FALSE;
	HOME_2STEP := 1;
	bAutoHomeOnly45 := TRUE;
END_IF

IF (一键回原点 AND PLC_Ready AND ((PLC_Deploy_State=0) OR (PLC_Deploy_State=30))) OR bAutoHomeReq THEN
	// Scraper/photo sequence is manual-only: 10Z, then 9X and 8Y.
	CASE HOME_1STEP OF
		1:
			IF 刮板轴10ZDATE.bHomed THEN
				刮板轴9XDATE.bHomed := FALSE; 刮板轴9XDATE.xHome := TRUE;
				拍照轴8YDATE.bHomed := FALSE; 拍照轴8YDATE.xHome := TRUE;
				HOME_1STEP := 2;
			END_IF
		2:
			IF 刮板轴10ZDATE.bHomed AND 刮板轴9XDATE.bHomed AND 拍照轴8YDATE.bHomed THEN
				HOME_1STEP := 0;
			END_IF
	END_CASE

	// Sampling sequence: 5Z retreat -> 5Z home -> 4X retreat -> 4X home.
	CASE HOME_2STEP OF
		1:
			上样轴5Z轴DATE.xHome := FALSE;
			上样轴4X轴DATE.xHome := FALSE;
			上样轴5Z轴DATE.xMoveRel := FALSE;
			上样轴4X轴DATE.xMoveRel := FALSE;
			// Positive retreat is the established mechanical direction.  Do not
			// arm it when the positive hardware/software limit says that direction
			// is unavailable; the startup FSM reports the specific step failure.
			IF NOT b5ZRetreatUnsafe THEN
				HOME_2STEP := 2;
			END_IF
		2:
			上样轴5Z轴DATE.fRelTarget := 10.0;
			上样轴5Z轴DATE.fVelocity := 5.0;
			上样轴5Z轴DATE.xMoveRel := TRUE;
			HOME_2STEP := 3;
		3:
			上样轴5Z轴DATE.fRelTarget := 10.0;
			上样轴5Z轴DATE.fVelocity := 5.0;
			上样轴5Z轴DATE.xMoveRel := TRUE;
			IF 上样轴5Z轴DATE.bReMoveDone THEN
				上样轴5Z轴DATE.xMoveRel := FALSE;
				上样轴5Z轴DATE.bHomed := FALSE;
				上样轴5Z轴DATE.xHome := TRUE;
				HOME_2STEP := 4;
			END_IF
		4:
			上样轴5Z轴DATE.xHome := TRUE;
			IF 上样轴5Z轴DATE.bHomed THEN
				上样轴5Z轴DATE.xHome := FALSE;
				IF NOT bAutoHomeOnly45 THEN
					打样瓶上料轴3YDATE.bHomed := FALSE;
					打样瓶上料轴3YDATE.xHome := TRUE;
				END_IF
				IF (上样轴5Z轴DATE.fActPos < 3) AND NOT b4XRetreatUnsafe THEN
					上样轴4X轴DATE.fRelTarget := 10.0;
					上样轴4X轴DATE.fVelocity := 5.0;
					上样轴4X轴DATE.xMoveRel := TRUE;
					HOME_2STEP := 5;
				END_IF
			END_IF
		5:
			上样轴4X轴DATE.fRelTarget := 10.0;
			上样轴4X轴DATE.fVelocity := 5.0;
			上样轴4X轴DATE.xMoveRel := TRUE;
			IF 上样轴4X轴DATE.bReMoveDone THEN
				上样轴4X轴DATE.xMoveRel := FALSE;
				上样轴4X轴DATE.bHomed := FALSE;
				上样轴4X轴DATE.xHome := TRUE;
				HOME_2STEP := 6;
			END_IF
		6:
			上样轴4X轴DATE.xHome := TRUE;
			IF (bAutoHomeOnly45 OR 打样瓶上料轴3YDATE.bHomed) AND 上样轴4X轴DATE.bHomed THEN
				上样轴4X轴DATE.xHome := FALSE;
				HOME_2STEP := 0;
			END_IF
	END_CASE
END_IF

IF 玻璃上料轴1ZDATE.bHomed AND 玻璃上料轴2ZDATE.bHomed AND 点样轴6XDATE.bHomed
	AND 点样轴7YDATE.bHomed AND 地轨轴11YDATE.bHomed AND 刮板轴10ZDATE.bHomed
	AND 刮板轴9XDATE.bHomed AND 上样轴5Z轴DATE.bHomed AND 上样轴4X轴DATE.bHomed
	AND 拍照轴8YDATE.bHomed AND 打样瓶上料轴3YDATE.bHomed THEN
	一键回原点 := FALSE;
END_IF
END_ACTION

ACTION 伺服调用:
//玻璃上料轴1Z伺服控制
FB_SERVOAXIS_0(
	AXIS:= 玻璃上料轴1Z ,                    //轴名称
	xEnable:=急停  ,                         //轴使能
	xStartupMotionAllowed:= FALSE, // startup axis ownership
	xHome:= 玻璃上料轴1ZDATE.xHome,          //轴回零命令
	xJogPos:=玻璃上料轴1ZDATE.xJogPos OR Z1JOG_pos  ,     //轴正转命令
	xJogNeg:=玻璃上料轴1ZDATE.xJogNeg OR Z1JOG_neg ,     //轴反转命令
	xStop:= 玻璃上料轴1ZDATE.xStop ,         //轴停止命令
	xMoveAbs:= 玻璃上料轴1ZDATE.xMoveAbs ,   //轴绝对定位命令
	xMoveRel:= 玻璃上料轴1ZDATE.xMoveRel,    //轴相对定位命令
	XReset:= 玻璃上料轴1ZDATE.XReset OR 复位 OR bSysReset ,       //轴复位
	fAbsTarget:= 玻璃上料轴1ZDATE.fAbsTarget ,  //轴绝对定位距离
	fRelTarget:=玻璃上料轴1ZDATE.fRelTarget  ,  //轴相对移动距离
	fVelocity:= 玻璃上料轴1ZDATE.fVelocity ,    //轴定位速度
	fAcc:=1000.0 ,              //轴加速度
	fDec:= 1000.0,              //轴减速度
	fJogVel:= 15.0 ,        //轴JOG速度
	bEnabled=> 玻璃上料轴1ZDATE.bEnabled ,      //轴使能完成
	bHomed=> 回零完成1Z ,          //轴回原点完成
	bBusy=> 玻璃上料轴1ZDATE.bBusy ,            //轴运行中
	fActPos=>玻璃上料轴1ZDATE.fActPos  ,        //轴当前位置
	fActVel=>玻璃上料轴1ZDATE.fActVel  ,        //轴当前速度
	bAbMoveDone=>玻璃上料轴1ZDATE.bAbMoveDone ,  //轴绝对定位完成
	bReMoveDone =>玻璃上料轴1ZDATE.bReMoveDone ,);    //轴相对定位完成 
// startup alarm visibility axis 0
玻璃上料轴1ZDATE.bError := FB_SERVOAXIS_0.bError AND NOT PLC_Startup_AlarmInhibit;
IF PLC_Startup_AlarmInhibit THEN
	玻璃上料轴1ZDATE.iErrorCode := 0;
ELSE
	玻璃上料轴1ZDATE.iErrorCode := FB_SERVOAXIS_0.iErrorCode;
END_IF
IF 回零完成1Z THEN
	玻璃上料轴1ZDATE.xHome := FALSE;
	玻璃上料轴1ZDATE.bHomed := TRUE;
END_IF

//玻璃上料轴2Z伺服控制
FB_SERVOAXIS_1(
	AXIS:= 玻璃上料轴2Z ,                    //轴名称
	xEnable:=急停  ,                         //轴使能
	xStartupMotionAllowed:= FALSE, // startup axis ownership
	xHome:= 玻璃上料轴2ZDATE.xHome,          //轴回零命令
	xJogPos:=玻璃上料轴2ZDATE.xJogPos OR Z2JOG_POS ,     //轴正转命令
	xJogNeg:=玻璃上料轴2ZDATE.xJogNeg OR Z2JOG_NEG ,     //轴反转命令
	xStop:= 玻璃上料轴2ZDATE.xStop ,         //轴停止命令
	xMoveAbs:= 玻璃上料轴2ZDATE.xMoveAbs ,   //轴绝对定位命令
	xMoveRel:= 玻璃上料轴2ZDATE.xMoveRel,    //轴相对定位命令
	XReset:= 玻璃上料轴2ZDATE.XReset OR 复位 OR bSysReset ,       //轴复位
	fAbsTarget:= 玻璃上料轴2ZDATE.fAbsTarget ,  //轴绝对定位距离
	fRelTarget:=玻璃上料轴2ZDATE.fRelTarget  ,  //轴相对移动距离
	fVelocity:= 玻璃上料轴2ZDATE.fVelocity ,    //轴定位速度
	fAcc:=1000.0 ,              //轴加速度
	fDec:= 1000.0,              //轴减速度
	fJogVel:= 15.0 ,        //轴JOG速度
	bEnabled=> 玻璃上料轴2ZDATE.bEnabled ,      //轴使能完成
	bHomed=> 回零完成2Z ,          //轴回原点完成
	bBusy=> 玻璃上料轴2ZDATE.bBusy ,            //轴运行中
	fActPos=>玻璃上料轴2ZDATE.fActPos  ,        //轴当前位置
	fActVel=>玻璃上料轴2ZDATE.fActVel  ,        //轴当前速度
	bAbMoveDone=>玻璃上料轴2ZDATE.bAbMoveDone ,  //轴绝对定位完成
	bReMoveDone =>玻璃上料轴2ZDATE.bReMoveDone ,);    //轴相对定位完成 
// startup alarm visibility axis 1
玻璃上料轴2ZDATE.bError := FB_SERVOAXIS_1.bError AND NOT PLC_Startup_AlarmInhibit;
IF PLC_Startup_AlarmInhibit THEN
	玻璃上料轴2ZDATE.iErrorCode := 0;
ELSE
	玻璃上料轴2ZDATE.iErrorCode := FB_SERVOAXIS_1.iErrorCode;
END_IF
IF 回零完成2Z THEN
	玻璃上料轴2ZDATE.xHome := FALSE;
	玻璃上料轴2ZDATE.bHomed := TRUE;
END_IF	
	
FB_SERVOAXIS_2(
	AXIS:= 打样瓶上料轴3Y ,                    //轴名称
	xEnable:= 急停 AND NOT (Sampling_Servo_FreeMove AND (上样轴5Z轴DATE.fActPos < 3)) ,   //轴使能(去使能手推: 仅5Z抬起<3时放开3Y)
	xStartupMotionAllowed:= FALSE, // startup axis ownership
	xHome:= 打样瓶上料轴3YDATE.xHome,          //轴回零命令
	xJogPos:=打样瓶上料轴3YDATE.xJogPos  ,     //轴正转命令
	xJogNeg:=打样瓶上料轴3YDATE.xJogNeg  ,     //轴反转命令
	xStop:= 打样瓶上料轴3YDATE.xStop ,         //轴停止命令
	xMoveAbs:= 打样瓶上料轴3YDATE.xMoveAbs ,   //轴绝对定位命令
	xMoveRel:= 打样瓶上料轴3YDATE.xMoveRel,    //轴相对定位命令
	XReset:= 打样瓶上料轴3YDATE.XReset OR 复位 OR bSysReset,       //轴复位
	fAbsTarget:= 打样瓶上料轴3YDATE.fAbsTarget ,  //轴绝对定位距离
	fRelTarget:=打样瓶上料轴3YDATE.fRelTarget  ,  //轴相对移动距离
	fVelocity:= 打样瓶上料轴3YDATE.fVelocity ,    //轴定位速度
	fAcc:=500.0 ,              //轴加速度
	fDec:= 500.0 ,              //轴减速度
	fJogVel:= 50.0 ,        //轴JOG速度
	bEnabled=> 打样瓶上料轴3YDATE.bEnabled ,      //轴使能完成
	bHomed=> 回零完成3Y ,          //轴回原点完成
	bBusy=> 打样瓶上料轴3YDATE.bBusy ,            //轴运行中
	fActPos=>打样瓶上料轴3YDATE.fActPos  ,        //轴当前位置
	fActVel=>打样瓶上料轴3YDATE.fActVel  ,        //轴当前速度
	bAbMoveDone=>打样瓶上料轴3YDATE.bAbMoveDone ,  //轴绝对定位完成
	bReMoveDone =>打样瓶上料轴3YDATE.bReMoveDone ,);    //轴相对定位完成 
// startup alarm visibility axis 2
打样瓶上料轴3YDATE.bError := FB_SERVOAXIS_2.bError AND NOT PLC_Startup_AlarmInhibit;
IF PLC_Startup_AlarmInhibit THEN
	打样瓶上料轴3YDATE.iErrorCode := 0;
ELSE
	打样瓶上料轴3YDATE.iErrorCode := FB_SERVOAXIS_2.iErrorCode;
END_IF
IF 回零完成3Y THEN
	打样瓶上料轴3YDATE.xHome := FALSE;
	打样瓶上料轴3YDATE.bHomed := TRUE;
END_IF		

